(* Logix 5000 project; controller reports 1756-L63 rev 20.15; software revision 20.04; part 6 of 52 *)

        [520].time.Hour := 2, [520].time.Minute := 29, [520].time.Second := 59, [521].log_data[0].min := 1.0, [521].log_data[0].max := 1.0, [521].log_data[0].total := 900.0, [521].log_data[0].time := 900.0, [521].log_data[0].minminute := 30, [521].log_data[0].maxminute := 30, [521].log_data[0].valid := 1, [521].log_data[1].valid := 1, [521].log_data[2].valid := 1, [521].log_data[3].valid := 1, [521].log_data[4].valid := 1, [521].log_data[5].valid := 1, [521].log_data[6].valid := 1, [521].log_data[7].valid := 1, [521].log_data[8].valid := 1, [521].log_data[9].valid := 1, [521].log_data[10].valid := 1, [521].log_data[11].valid := 1, [521].log_data[12].valid := 1, [521].log_data[13].valid := 1, [521].log_data[14].valid := 1, [521].log_data[15].valid := 1, [521].log_data[16].valid := 1, [521].log_data[17].valid := 1, [521].log_data[18].valid := 1, [521].log_data[19].valid := 1, [521].time.Year := 2023, [521].time.Month := 1, [521].time.Day := 13, [521].time.Hour := 2, [521].time.Minute := 44, [521].time.Second := 59, [522].log_data[0].min := 1.0, [522].log_data[0].max := 1.0, [522].log_data[0].total := 900.0, [522].log_data[0].time := 900.0, [522].log_data[0].minminute := 45, [522].log_data[0].maxminute := 45, [522].log_data[0].valid := 1, [522].log_data[1].valid := 1, [522].log_data[2].valid := 1, [522].log_data[3].valid := 1, [522].log_data[4].valid := 1, [522].log_data[5].valid := 1, [522].log_data[6].valid := 1, [522].log_data[7].valid := 1, [522].log_data[8].valid := 1, [522].log_data[9].valid := 1, [522].log_data[10].valid := 1, [522].log_data[11].valid := 1, [522].log_data[12].valid := 1, [522].log_data[13].valid := 1, [522].log_data[14].valid := 1, [522].log_data[15].valid := 1, [522].log_data[16].valid := 1, [522].log_data[17].valid := 1, [522].log_data[18].valid := 1,
        [522].log_data[19].valid := 1, [522].time.Year := 2023, [522].time.Month := 1, [522].time.Day := 13, [522].time.Hour := 2, [522].time.Minute := 59, [522].time.Second := 59, [523].log_data[0].min := 1.0, [523].log_data[0].max := 1.0, [523].log_data[0].total := 900.0, [523].log_data[0].time := 900.0, [523].log_data[0].valid := 1, [523].log_data[1].valid := 1, [523].log_data[2].valid := 1, [523].log_data[3].valid := 1, [523].log_data[4].valid := 1, [523].log_data[5].valid := 1, [523].log_data[6].valid := 1, [523].log_data[7].valid := 1, [523].log_data[8].valid := 1, [523].log_data[9].valid := 1, [523].log_data[10].valid := 1, [523].log_data[11].valid := 1, [523].log_data[12].valid := 1, [523].log_data[13].valid := 1, [523].log_data[14].valid := 1, [523].log_data[15].valid := 1, [523].log_data[16].valid := 1, [523].log_data[17].valid := 1, [523].log_data[18].valid := 1, [523].log_data[19].valid := 1, [523].time.Year := 2023, [523].time.Month := 1, [523].time.Day := 13, [523].time.Hour := 3, [523].time.Minute := 14, [523].time.Second := 59, [524].log_data[0].min := 1.0, [524].log_data[0].max := 1.0, [524].log_data[0].total := 900.0, [524].log_data[0].time := 900.0, [524].log_data[0].minminute := 15, [524].log_data[0].maxminute := 15, [524].log_data[0].valid := 1, [524].log_data[1].valid := 1, [524].log_data[2].valid := 1, [524].log_data[3].valid := 1, [524].log_data[4].valid := 1, [524].log_data[5].valid := 1, [524].log_data[6].valid := 1, [524].log_data[7].valid := 1, [524].log_data[8].valid := 1, [524].log_data[9].valid := 1, [524].log_data[10].valid := 1, [524].log_data[11].valid := 1, [524].log_data[12].valid := 1, [524].log_data[13].valid := 1, [524].log_data[14].valid := 1, [524].log_data[15].valid := 1, [524].log_data[16].valid := 1,
        [524].log_data[17].valid := 1, [524].log_data[18].valid := 1, [524].log_data[19].valid := 1, [524].time.Year := 2023, [524].time.Month := 1, [524].time.Day := 13, [524].time.Hour := 3, [524].time.Minute := 29, [524].time.Second := 59, [525].log_data[0].min := 1.0, [525].log_data[0].max := 1.0, [525].log_data[0].total := 900.0, [525].log_data[0].time := 900.0, [525].log_data[0].minminute := 30, [525].log_data[0].maxminute := 30, [525].log_data[0].valid := 1, [525].log_data[1].valid := 1, [525].log_data[2].valid := 1, [525].log_data[3].valid := 1, [525].log_data[4].valid := 1, [525].log_data[5].valid := 1, [525].log_data[6].valid := 1, [525].log_data[7].valid := 1, [525].log_data[8].valid := 1, [525].log_data[9].valid := 1, [525].log_data[10].valid := 1, [525].log_data[11].valid := 1, [525].log_data[12].valid := 1, [525].log_data[13].valid := 1, [525].log_data[14].valid := 1, [525].log_data[15].valid := 1, [525].log_data[16].valid := 1, [525].log_data[17].valid := 1, [525].log_data[18].valid := 1, [525].log_data[19].valid := 1, [525].time.Year := 2023, [525].time.Month := 1, [525].time.Day := 13, [525].time.Hour := 3, [525].time.Minute := 44, [525].time.Second := 59, [526].log_data[0].min := 1.0, [526].log_data[0].max := 1.0, [526].log_data[0].total := 900.0, [526].log_data[0].time := 900.0, [526].log_data[0].minminute := 45, [526].log_data[0].maxminute := 45, [526].log_data[0].valid := 1, [526].log_data[1].valid := 1, [526].log_data[2].valid := 1, [526].log_data[3].valid := 1, [526].log_data[4].valid := 1, [526].log_data[5].valid := 1, [526].log_data[6].valid := 1, [526].log_data[7].valid := 1, [526].log_data[8].valid := 1, [526].log_data[9].valid := 1, [526].log_data[10].valid := 1, [526].log_data[11].valid := 1, [526].log_data[12].valid := 1,
        [526].log_data[13].valid := 1, [526].log_data[14].valid := 1, [526].log_data[15].valid := 1, [526].log_data[16].valid := 1, [526].log_data[17].valid := 1, [526].log_data[18].valid := 1, [526].log_data[19].valid := 1, [526].time.Year := 2023, [526].time.Month := 1, [526].time.Day := 13, [526].time.Hour := 3, [526].time.Minute := 59, [526].time.Second := 59, [527].log_data[0].min := 1.0, [527].log_data[0].max := 1.0, [527].log_data[0].total := 900.0, [527].log_data[0].time := 900.0, [527].log_data[0].valid := 1, [527].log_data[1].valid := 1, [527].log_data[2].valid := 1, [527].log_data[3].valid := 1, [527].log_data[4].valid := 1, [527].log_data[5].valid := 1, [527].log_data[6].valid := 1, [527].log_data[7].valid := 1, [527].log_data[8].valid := 1, [527].log_data[9].valid := 1, [527].log_data[10].valid := 1, [527].log_data[11].valid := 1, [527].log_data[12].valid := 1, [527].log_data[13].valid := 1, [527].log_data[14].valid := 1, [527].log_data[15].valid := 1, [527].log_data[16].valid := 1, [527].log_data[17].valid := 1, [527].log_data[18].valid := 1, [527].log_data[19].valid := 1, [527].time.Year := 2023, [527].time.Month := 1, [527].time.Day := 13, [527].time.Hour := 4, [527].time.Minute := 14, [527].time.Second := 59, [528].log_data[0].min := 1.0, [528].log_data[0].max := 1.0, [528].log_data[0].total := 900.0, [528].log_data[0].time := 900.0, [528].log_data[0].minminute := 15, [528].log_data[0].maxminute := 15, [528].log_data[0].valid := 1, [528].log_data[1].valid := 1, [528].log_data[2].valid := 1, [528].log_data[3].valid := 1, [528].log_data[4].valid := 1, [528].log_data[5].valid := 1, [528].log_data[6].valid := 1, [528].log_data[7].valid := 1, [528].log_data[8].valid := 1, [528].log_data[9].valid := 1, [528].log_data[10].valid := 1,
        [528].log_data[11].valid := 1, [528].log_data[12].valid := 1, [528].log_data[13].valid := 1, [528].log_data[14].valid := 1, [528].log_data[15].valid := 1, [528].log_data[16].valid := 1, [528].log_data[17].valid := 1, [528].log_data[18].valid := 1, [528].log_data[19].valid := 1, [528].time.Year := 2023, [528].time.Month := 1, [528].time.Day := 13, [528].time.Hour := 4, [528].time.Minute := 29, [528].time.Second := 59, [529].log_data[0].min := 1.0, [529].log_data[0].max := 1.0, [529].log_data[0].total := 900.0, [529].log_data[0].time := 900.0, [529].log_data[0].minminute := 30, [529].log_data[0].maxminute := 30, [529].log_data[0].valid := 1, [529].log_data[1].valid := 1, [529].log_data[2].valid := 1, [529].log_data[3].valid := 1, [529].log_data[4].valid := 1, [529].log_data[5].valid := 1, [529].log_data[6].valid := 1, [529].log_data[7].valid := 1, [529].log_data[8].valid := 1, [529].log_data[9].valid := 1, [529].log_data[10].valid := 1, [529].log_data[11].valid := 1, [529].log_data[12].valid := 1, [529].log_data[13].valid := 1, [529].log_data[14].valid := 1, [529].log_data[15].valid := 1, [529].log_data[16].valid := 1, [529].log_data[17].valid := 1, [529].log_data[18].valid := 1, [529].log_data[19].valid := 1, [529].time.Year := 2023, [529].time.Month := 1, [529].time.Day := 13, [529].time.Hour := 4, [529].time.Minute := 44, [529].time.Second := 59, [530].log_data[0].min := 1.0, [530].log_data[0].max := 1.0, [530].log_data[0].total := 900.0, [530].log_data[0].time := 900.0, [530].log_data[0].minminute := 45, [530].log_data[0].maxminute := 45, [530].log_data[0].valid := 1, [530].log_data[1].valid := 1, [530].log_data[2].valid := 1, [530].log_data[3].valid := 1, [530].log_data[4].valid := 1, [530].log_data[5].valid := 1, [530].log_data[6].valid := 1,
        [530].log_data[7].valid := 1, [530].log_data[8].valid := 1, [530].log_data[9].valid := 1, [530].log_data[10].valid := 1, [530].log_data[11].valid := 1, [530].log_data[12].valid := 1, [530].log_data[13].valid := 1, [530].log_data[14].valid := 1, [530].log_data[15].valid := 1, [530].log_data[16].valid := 1, [530].log_data[17].valid := 1, [530].log_data[18].valid := 1, [530].log_data[19].valid := 1, [530].time.Year := 2023, [530].time.Month := 1, [530].time.Day := 13, [530].time.Hour := 4, [530].time.Minute := 59, [530].time.Second := 59, [531].log_data[0].min := 1.0, [531].log_data[0].max := 1.0, [531].log_data[0].total := 900.0, [531].log_data[0].time := 900.0, [531].log_data[0].valid := 1, [531].log_data[1].valid := 1, [531].log_data[2].valid := 1, [531].log_data[3].valid := 1, [531].log_data[4].valid := 1, [531].log_data[5].valid := 1, [531].log_data[6].valid := 1, [531].log_data[7].valid := 1, [531].log_data[8].valid := 1, [531].log_data[9].valid := 1, [531].log_data[10].valid := 1, [531].log_data[11].valid := 1, [531].log_data[12].valid := 1, [531].log_data[13].valid := 1, [531].log_data[14].valid := 1, [531].log_data[15].valid := 1, [531].log_data[16].valid := 1, [531].log_data[17].valid := 1, [531].log_data[18].valid := 1, [531].log_data[19].valid := 1, [531].time.Year := 2023, [531].time.Month := 1, [531].time.Day := 13, [531].time.Hour := 5, [531].time.Minute := 14, [531].time.Second := 59, [532].log_data[0].min := 1.0, [532].log_data[0].max := 1.0, [532].log_data[0].total := 900.0, [532].log_data[0].time := 900.0, [532].log_data[0].minminute := 15, [532].log_data[0].maxminute := 15, [532].log_data[0].valid := 1, [532].log_data[1].valid := 1, [532].log_data[2].valid := 1, [532].log_data[3].valid := 1, [532].log_data[4].valid := 1,
        [532].log_data[5].valid := 1, [532].log_data[6].valid := 1, [532].log_data[7].valid := 1, [532].log_data[8].valid := 1, [532].log_data[9].valid := 1, [532].log_data[10].valid := 1, [532].log_data[11].valid := 1, [532].log_data[12].valid := 1, [532].log_data[13].valid := 1, [532].log_data[14].valid := 1, [532].log_data[15].valid := 1, [532].log_data[16].valid := 1, [532].log_data[17].valid := 1, [532].log_data[18].valid := 1, [532].log_data[19].valid := 1, [532].time.Year := 2023, [532].time.Month := 1, [532].time.Day := 13, [532].time.Hour := 5, [532].time.Minute := 29, [532].time.Second := 59, [533].log_data[0].min := 1.0, [533].log_data[0].max := 1.0, [533].log_data[0].total := 900.0, [533].log_data[0].time := 900.0, [533].log_data[0].minminute := 30, [533].log_data[0].maxminute := 30, [533].log_data[0].valid := 1, [533].log_data[1].valid := 1, [533].log_data[2].valid := 1, [533].log_data[3].valid := 1, [533].log_data[4].valid := 1, [533].log_data[5].valid := 1, [533].log_data[6].valid := 1, [533].log_data[7].valid := 1, [533].log_data[8].valid := 1, [533].log_data[9].valid := 1, [533].log_data[10].valid := 1, [533].log_data[11].valid := 1, [533].log_data[12].valid := 1, [533].log_data[13].valid := 1, [533].log_data[14].valid := 1, [533].log_data[15].valid := 1, [533].log_data[16].valid := 1, [533].log_data[17].valid := 1, [533].log_data[18].valid := 1, [533].log_data[19].valid := 1, [533].time.Year := 2023, [533].time.Month := 1, [533].time.Day := 13, [533].time.Hour := 5, [533].time.Minute := 44, [533].time.Second := 59, [534].log_data[0].min := 1.0, [534].log_data[0].max := 1.0, [534].log_data[0].total := 900.0, [534].log_data[0].time := 900.0, [534].log_data[0].minminute := 45, [534].log_data[0].maxminute := 45, [534].log_data[0].valid := 1,
        [534].log_data[1].valid := 1, [534].log_data[2].valid := 1, [534].log_data[3].valid := 1, [534].log_data[4].valid := 1, [534].log_data[5].valid := 1, [534].log_data[6].valid := 1, [534].log_data[7].valid := 1, [534].log_data[8].valid := 1, [534].log_data[9].valid := 1, [534].log_data[10].valid := 1, [534].log_data[11].valid := 1, [534].log_data[12].valid := 1, [534].log_data[13].valid := 1, [534].log_data[14].valid := 1, [534].log_data[15].valid := 1, [534].log_data[16].valid := 1, [534].log_data[17].valid := 1, [534].log_data[18].valid := 1, [534].log_data[19].valid := 1, [534].time.Year := 2023, [534].time.Month := 1, [534].time.Day := 13, [534].time.Hour := 5, [534].time.Minute := 59, [534].time.Second := 59, [535].log_data[0].min := 1.0, [535].log_data[0].max := 1.0, [535].log_data[0].total := 900.0, [535].log_data[0].time := 900.0, [535].log_data[0].valid := 1, [535].log_data[1].valid := 1, [535].log_data[2].valid := 1, [535].log_data[3].valid := 1, [535].log_data[4].valid := 1, [535].log_data[5].valid := 1, [535].log_data[6].valid := 1, [535].log_data[7].valid := 1, [535].log_data[8].valid := 1, [535].log_data[9].valid := 1, [535].log_data[10].valid := 1, [535].log_data[11].valid := 1, [535].log_data[12].valid := 1, [535].log_data[13].valid := 1, [535].log_data[14].valid := 1, [535].log_data[15].valid := 1, [535].log_data[16].valid := 1, [535].log_data[17].valid := 1, [535].log_data[18].valid := 1, [535].log_data[19].valid := 1, [535].time.Year := 2023, [535].time.Month := 1, [535].time.Day := 13, [535].time.Hour := 6, [535].time.Minute := 14, [535].time.Second := 59, [536].log_data[0].min := 1.0, [536].log_data[0].max := 1.0, [536].log_data[0].total := 900.0, [536].log_data[0].time := 900.0, [536].log_data[0].minminute := 15,
        [536].log_data[0].maxminute := 15, [536].log_data[0].valid := 1, [536].log_data[1].valid := 1, [536].log_data[2].valid := 1, [536].log_data[3].valid := 1, [536].log_data[4].valid := 1, [536].log_data[5].valid := 1, [536].log_data[6].valid := 1, [536].log_data[7].valid := 1, [536].log_data[8].valid := 1, [536].log_data[9].valid := 1, [536].log_data[10].valid := 1, [536].log_data[11].valid := 1, [536].log_data[12].valid := 1, [536].log_data[13].valid := 1, [536].log_data[14].valid := 1, [536].log_data[15].valid := 1, [536].log_data[16].valid := 1, [536].log_data[17].valid := 1, [536].log_data[18].valid := 1, [536].log_data[19].valid := 1, [536].time.Year := 2023, [536].time.Month := 1, [536].time.Day := 13, [536].time.Hour := 6, [536].time.Minute := 29, [536].time.Second := 59, [537].log_data[0].min := 1.0, [537].log_data[0].max := 1.0, [537].log_data[0].total := 900.0, [537].log_data[0].time := 900.0, [537].log_data[0].minminute := 30, [537].log_data[0].maxminute := 30, [537].log_data[0].valid := 1, [537].log_data[1].valid := 1, [537].log_data[2].valid := 1, [537].log_data[3].valid := 1, [537].log_data[4].valid := 1, [537].log_data[5].valid := 1, [537].log_data[6].valid := 1, [537].log_data[7].valid := 1, [537].log_data[8].valid := 1, [537].log_data[9].valid := 1, [537].log_data[10].valid := 1, [537].log_data[11].valid := 1, [537].log_data[12].valid := 1, [537].log_data[13].valid := 1, [537].log_data[14].valid := 1, [537].log_data[15].valid := 1, [537].log_data[16].valid := 1, [537].log_data[17].valid := 1, [537].log_data[18].valid := 1, [537].log_data[19].valid := 1, [537].time.Year := 2023, [537].time.Month := 1, [537].time.Day := 13, [537].time.Hour := 6, [537].time.Minute := 44, [537].time.Second := 59, [538].log_data[0].min := 1.0,
        [538].log_data[0].max := 1.0, [538].log_data[0].total := 900.0, [538].log_data[0].time := 900.0, [538].log_data[0].minminute := 45, [538].log_data[0].maxminute := 45, [538].log_data[0].valid := 1, [538].log_data[1].valid := 1, [538].log_data[2].valid := 1, [538].log_data[3].valid := 1, [538].log_data[4].valid := 1, [538].log_data[5].valid := 1, [538].log_data[6].valid := 1, [538].log_data[7].valid := 1, [538].log_data[8].valid := 1, [538].log_data[9].valid := 1, [538].log_data[10].valid := 1, [538].log_data[11].valid := 1, [538].log_data[12].valid := 1, [538].log_data[13].valid := 1, [538].log_data[14].valid := 1, [538].log_data[15].valid := 1, [538].log_data[16].valid := 1, [538].log_data[17].valid := 1, [538].log_data[18].valid := 1, [538].log_data[19].valid := 1, [538].time.Year := 2023, [538].time.Month := 1, [538].time.Day := 13, [538].time.Hour := 6, [538].time.Minute := 59, [538].time.Second := 59, [539].log_data[0].min := 1.0, [539].log_data[0].max := 1.0, [539].log_data[0].total := 900.0, [539].log_data[0].time := 900.0, [539].log_data[0].valid := 1, [539].log_data[1].valid := 1, [539].log_data[2].valid := 1, [539].log_data[3].valid := 1, [539].log_data[4].valid := 1, [539].log_data[5].valid := 1, [539].log_data[6].valid := 1, [539].log_data[7].valid := 1, [539].log_data[8].valid := 1, [539].log_data[9].valid := 1, [539].log_data[10].valid := 1, [539].log_data[11].valid := 1, [539].log_data[12].valid := 1, [539].log_data[13].valid := 1, [539].log_data[14].valid := 1, [539].log_data[15].valid := 1, [539].log_data[16].valid := 1, [539].log_data[17].valid := 1, [539].log_data[18].valid := 1, [539].log_data[19].valid := 1, [539].time.Year := 2023, [539].time.Month := 1, [539].time.Day := 13, [539].time.Hour := 7, [539].time.Minute := 14,
        [539].time.Second := 59, [540].log_data[0].min := 1.0, [540].log_data[0].max := 1.0, [540].log_data[0].total := 900.0, [540].log_data[0].time := 900.0, [540].log_data[0].minminute := 15, [540].log_data[0].maxminute := 15, [540].log_data[0].valid := 1, [540].log_data[1].valid := 1, [540].log_data[2].valid := 1, [540].log_data[3].valid := 1, [540].log_data[4].valid := 1, [540].log_data[5].valid := 1, [540].log_data[6].valid := 1, [540].log_data[7].valid := 1, [540].log_data[8].valid := 1, [540].log_data[9].valid := 1, [540].log_data[10].valid := 1, [540].log_data[11].valid := 1, [540].log_data[12].valid := 1, [540].log_data[13].valid := 1, [540].log_data[14].valid := 1, [540].log_data[15].valid := 1, [540].log_data[16].valid := 1, [540].log_data[17].valid := 1, [540].log_data[18].valid := 1, [540].log_data[19].valid := 1, [540].time.Year := 2023, [540].time.Month := 1, [540].time.Day := 13, [540].time.Hour := 7, [540].time.Minute := 29, [540].time.Second := 59, [541].log_data[0].min := 1.0, [541].log_data[0].max := 1.0, [541].log_data[0].total := 900.0, [541].log_data[0].time := 900.0, [541].log_data[0].minminute := 30, [541].log_data[0].maxminute := 30, [541].log_data[0].valid := 1, [541].log_data[1].valid := 1, [541].log_data[2].valid := 1, [541].log_data[3].valid := 1, [541].log_data[4].valid := 1, [541].log_data[5].valid := 1, [541].log_data[6].valid := 1, [541].log_data[7].valid := 1, [541].log_data[8].valid := 1, [541].log_data[9].valid := 1, [541].log_data[10].valid := 1, [541].log_data[11].valid := 1, [541].log_data[12].valid := 1, [541].log_data[13].valid := 1, [541].log_data[14].valid := 1, [541].log_data[15].valid := 1, [541].log_data[16].valid := 1, [541].log_data[17].valid := 1, [541].log_data[18].valid := 1, [541].log_data[19].valid := 1, [541].time.Year := 2023,
        [541].time.Month := 1, [541].time.Day := 13, [541].time.Hour := 7, [541].time.Minute := 44, [541].time.Second := 59, [542].log_data[0].min := 1.0, [542].log_data[0].max := 1.0, [542].log_data[0].total := 900.0, [542].log_data[0].time := 900.0, [542].log_data[0].minminute := 45, [542].log_data[0].maxminute := 45, [542].log_data[0].valid := 1, [542].log_data[1].valid := 1, [542].log_data[2].valid := 1, [542].log_data[3].valid := 1, [542].log_data[4].valid := 1, [542].log_data[5].valid := 1, [542].log_data[6].valid := 1, [542].log_data[7].valid := 1, [542].log_data[8].valid := 1, [542].log_data[9].valid := 1, [542].log_data[10].valid := 1, [542].log_data[11].valid := 1, [542].log_data[12].valid := 1, [542].log_data[13].valid := 1, [542].log_data[14].valid := 1, [542].log_data[15].valid := 1, [542].log_data[16].valid := 1, [542].log_data[17].valid := 1, [542].log_data[18].valid := 1, [542].log_data[19].valid := 1, [542].time.Year := 2023, [542].time.Month := 1, [542].time.Day := 13, [542].time.Hour := 7, [542].time.Minute := 59, [542].time.Second := 59, [543].log_data[0].min := 1.0, [543].log_data[0].max := 1.0, [543].log_data[0].total := 900.0, [543].log_data[0].time := 900.0, [543].log_data[0].valid := 1, [543].log_data[1].valid := 1, [543].log_data[2].valid := 1, [543].log_data[3].valid := 1, [543].log_data[4].valid := 1, [543].log_data[5].valid := 1, [543].log_data[6].valid := 1, [543].log_data[7].valid := 1, [543].log_data[8].valid := 1, [543].log_data[9].valid := 1, [543].log_data[10].valid := 1, [543].log_data[11].valid := 1, [543].log_data[12].valid := 1, [543].log_data[13].valid := 1, [543].log_data[14].valid := 1, [543].log_data[15].valid := 1, [543].log_data[16].valid := 1, [543].log_data[17].valid := 1, [543].log_data[18].valid := 1,
        [543].log_data[19].valid := 1, [543].time.Year := 2023, [543].time.Month := 1, [543].time.Day := 13, [543].time.Hour := 8, [543].time.Minute := 14, [543].time.Second := 59, [544].log_data[0].min := 1.0, [544].log_data[0].max := 1.0, [544].log_data[0].total := 900.0, [544].log_data[0].time := 900.0, [544].log_data[0].minminute := 15, [544].log_data[0].maxminute := 15, [544].log_data[0].valid := 1, [544].log_data[1].valid := 1, [544].log_data[2].valid := 1, [544].log_data[3].valid := 1, [544].log_data[4].valid := 1, [544].log_data[5].valid := 1, [544].log_data[6].valid := 1, [544].log_data[7].valid := 1, [544].log_data[8].valid := 1, [544].log_data[9].valid := 1, [544].log_data[10].valid := 1, [544].log_data[11].valid := 1, [544].log_data[12].valid := 1, [544].log_data[13].valid := 1, [544].log_data[14].valid := 1, [544].log_data[15].valid := 1, [544].log_data[16].valid := 1, [544].log_data[17].valid := 1, [544].log_data[18].valid := 1, [544].log_data[19].valid := 1, [544].time.Year := 2023, [544].time.Month := 1, [544].time.Day := 13, [544].time.Hour := 8, [544].time.Minute := 29, [544].time.Second := 59, [545].log_data[0].min := 1.0, [545].log_data[0].max := 1.0, [545].log_data[0].total := 900.0, [545].log_data[0].time := 900.0, [545].log_data[0].minminute := 30, [545].log_data[0].maxminute := 30, [545].log_data[0].valid := 1, [545].log_data[1].valid := 1, [545].log_data[2].valid := 1, [545].log_data[3].valid := 1, [545].log_data[4].valid := 1, [545].log_data[5].valid := 1, [545].log_data[6].valid := 1, [545].log_data[7].valid := 1, [545].log_data[8].valid := 1, [545].log_data[9].valid := 1, [545].log_data[10].valid := 1, [545].log_data[11].valid := 1, [545].log_data[12].valid := 1, [545].log_data[13].valid := 1, [545].log_data[14].valid := 1,
        [545].log_data[15].valid := 1, [545].log_data[16].valid := 1, [545].log_data[17].valid := 1, [545].log_data[18].valid := 1, [545].log_data[19].valid := 1, [545].time.Year := 2023, [545].time.Month := 1, [545].time.Day := 13, [545].time.Hour := 8, [545].time.Minute := 44, [545].time.Second := 59, [546].log_data[0].min := 1.0, [546].log_data[0].max := 1.0, [546].log_data[0].total := 900.0, [546].log_data[0].time := 900.0, [546].log_data[0].minminute := 45, [546].log_data[0].maxminute := 45, [546].log_data[0].valid := 1, [546].log_data[1].valid := 1, [546].log_data[2].valid := 1, [546].log_data[3].valid := 1, [546].log_data[4].valid := 1, [546].log_data[5].valid := 1, [546].log_data[6].valid := 1, [546].log_data[7].valid := 1, [546].log_data[8].valid := 1, [546].log_data[9].valid := 1, [546].log_data[10].valid := 1, [546].log_data[11].valid := 1, [546].log_data[12].valid := 1, [546].log_data[13].valid := 1, [546].log_data[14].valid := 1, [546].log_data[15].valid := 1, [546].log_data[16].valid := 1, [546].log_data[17].valid := 1, [546].log_data[18].valid := 1, [546].log_data[19].valid := 1, [546].time.Year := 2023, [546].time.Month := 1, [546].time.Day := 13, [546].time.Hour := 8, [546].time.Minute := 59, [546].time.Second := 59, [547].log_data[0].min := 1.0, [547].log_data[0].max := 1.0, [547].log_data[0].total := 900.0, [547].log_data[0].time := 900.0, [547].log_data[0].valid := 1, [547].log_data[1].valid := 1, [547].log_data[2].valid := 1, [547].log_data[3].valid := 1, [547].log_data[4].valid := 1, [547].log_data[5].valid := 1, [547].log_data[6].valid := 1, [547].log_data[7].valid := 1, [547].log_data[8].valid := 1, [547].log_data[9].valid := 1, [547].log_data[10].valid := 1, [547].log_data[11].valid := 1, [547].log_data[12].valid := 1,
        [547].log_data[13].valid := 1, [547].log_data[14].valid := 1, [547].log_data[15].valid := 1, [547].log_data[16].valid := 1, [547].log_data[17].valid := 1, [547].log_data[18].valid := 1, [547].log_data[19].valid := 1, [547].time.Year := 2023, [547].time.Month := 1, [547].time.Day := 13, [547].time.Hour := 9, [547].time.Minute := 14, [547].time.Second := 59, [548].log_data[0].min := 1.0, [548].log_data[0].max := 1.0, [548].log_data[0].total := 900.0, [548].log_data[0].time := 900.0, [548].log_data[0].minminute := 15, [548].log_data[0].maxminute := 15, [548].log_data[0].valid := 1, [548].log_data[1].valid := 1, [548].log_data[2].valid := 1, [548].log_data[3].valid := 1, [548].log_data[4].valid := 1, [548].log_data[5].valid := 1, [548].log_data[6].valid := 1, [548].log_data[7].valid := 1, [548].log_data[8].valid := 1, [548].log_data[9].valid := 1, [548].log_data[10].valid := 1, [548].log_data[11].valid := 1, [548].log_data[12].valid := 1, [548].log_data[13].valid := 1, [548].log_data[14].valid := 1, [548].log_data[15].valid := 1, [548].log_data[16].valid := 1, [548].log_data[17].valid := 1, [548].log_data[18].valid := 1, [548].log_data[19].valid := 1, [548].time.Year := 2023, [548].time.Month := 1, [548].time.Day := 13, [548].time.Hour := 9, [548].time.Minute := 29, [548].time.Second := 59, [549].log_data[0].min := 1.0, [549].log_data[0].max := 1.0, [549].log_data[0].total := 900.0, [549].log_data[0].time := 900.0, [549].log_data[0].minminute := 30, [549].log_data[0].maxminute := 30, [549].log_data[0].valid := 1, [549].log_data[1].valid := 1, [549].log_data[2].valid := 1, [549].log_data[3].valid := 1, [549].log_data[4].valid := 1, [549].log_data[5].valid := 1, [549].log_data[6].valid := 1, [549].log_data[7].valid := 1, [549].log_data[8].valid := 1,
        [549].log_data[9].valid := 1, [549].log_data[10].valid := 1, [549].log_data[11].valid := 1, [549].log_data[12].valid := 1, [549].log_data[13].valid := 1, [549].log_data[14].valid := 1, [549].log_data[15].valid := 1, [549].log_data[16].valid := 1, [549].log_data[17].valid := 1, [549].log_data[18].valid := 1, [549].log_data[19].valid := 1, [549].time.Year := 2023, [549].time.Month := 1, [549].time.Day := 13, [549].time.Hour := 9, [549].time.Minute := 44, [549].time.Second := 59, [550].log_data[0].min := 1.0, [550].log_data[0].max := 1.0, [550].log_data[0].total := 900.0, [550].log_data[0].time := 900.0, [550].log_data[0].minminute := 45, [550].log_data[0].maxminute := 45, [550].log_data[0].valid := 1, [550].log_data[1].valid := 1, [550].log_data[2].valid := 1, [550].log_data[3].valid := 1, [550].log_data[4].valid := 1, [550].log_data[5].valid := 1, [550].log_data[6].valid := 1, [550].log_data[7].valid := 1, [550].log_data[8].valid := 1, [550].log_data[9].valid := 1, [550].log_data[10].valid := 1, [550].log_data[11].valid := 1, [550].log_data[12].valid := 1, [550].log_data[13].valid := 1, [550].log_data[14].valid := 1, [550].log_data[15].valid := 1, [550].log_data[16].valid := 1, [550].log_data[17].valid := 1, [550].log_data[18].valid := 1, [550].log_data[19].valid := 1, [550].time.Year := 2023, [550].time.Month := 1, [550].time.Day := 13, [550].time.Hour := 9, [550].time.Minute := 59, [550].time.Second := 59, [551].log_data[0].min := 1.0, [551].log_data[0].max := 1.0, [551].log_data[0].total := 900.0, [551].log_data[0].time := 900.0, [551].log_data[0].valid := 1, [551].log_data[1].valid := 1, [551].log_data[2].valid := 1, [551].log_data[3].valid := 1, [551].log_data[4].valid := 1, [551].log_data[5].valid := 1, [551].log_data[6].valid := 1,
        [551].log_data[7].valid := 1, [551].log_data[8].valid := 1, [551].log_data[9].valid := 1, [551].log_data[10].valid := 1, [551].log_data[11].valid := 1, [551].log_data[12].valid := 1, [551].log_data[13].valid := 1, [551].log_data[14].valid := 1, [551].log_data[15].valid := 1, [551].log_data[16].valid := 1, [551].log_data[17].valid := 1, [551].log_data[18].valid := 1, [551].log_data[19].valid := 1, [551].time.Year := 2023, [551].time.Month := 1, [551].time.Day := 13, [551].time.Hour := 10, [551].time.Minute := 14, [551].time.Second := 59, [552].log_data[0].min := 1.0, [552].log_data[0].max := 1.0, [552].log_data[0].total := 900.0, [552].log_data[0].time := 900.0, [552].log_data[0].minminute := 15, [552].log_data[0].maxminute := 15, [552].log_data[0].valid := 1, [552].log_data[1].valid := 1, [552].log_data[2].valid := 1, [552].log_data[3].valid := 1, [552].log_data[4].valid := 1, [552].log_data[5].valid := 1, [552].log_data[6].valid := 1, [552].log_data[7].valid := 1, [552].log_data[8].valid := 1, [552].log_data[9].valid := 1, [552].log_data[10].valid := 1, [552].log_data[11].valid := 1, [552].log_data[12].valid := 1, [552].log_data[13].valid := 1, [552].log_data[14].valid := 1, [552].log_data[15].valid := 1, [552].log_data[16].valid := 1, [552].log_data[17].valid := 1, [552].log_data[18].valid := 1, [552].log_data[19].valid := 1, [552].time.Year := 2023, [552].time.Month := 1, [552].time.Day := 13, [552].time.Hour := 10, [552].time.Minute := 29, [552].time.Second := 59, [553].log_data[0].min := 1.0, [553].log_data[0].max := 1.0, [553].log_data[0].total := 900.0, [553].log_data[0].time := 900.0, [553].log_data[0].minminute := 30, [553].log_data[0].maxminute := 30, [553].log_data[0].valid := 1, [553].log_data[1].valid := 1, [553].log_data[2].valid := 1,
        [553].log_data[3].valid := 1, [553].log_data[4].valid := 1, [553].log_data[5].valid := 1, [553].log_data[6].valid := 1, [553].log_data[7].valid := 1, [553].log_data[8].valid := 1, [553].log_data[9].valid := 1, [553].log_data[10].valid := 1, [553].log_data[11].valid := 1, [553].log_data[12].valid := 1, [553].log_data[13].valid := 1, [553].log_data[14].valid := 1, [553].log_data[15].valid := 1, [553].log_data[16].valid := 1, [553].log_data[17].valid := 1, [553].log_data[18].valid := 1, [553].log_data[19].valid := 1, [553].time.Year := 2023, [553].time.Month := 1, [553].time.Day := 13, [553].time.Hour := 10, [553].time.Minute := 44, [553].time.Second := 59, [554].log_data[0].min := 1.0, [554].log_data[0].max := 1.0, [554].log_data[0].total := 900.0, [554].log_data[0].time := 900.0, [554].log_data[0].minminute := 45, [554].log_data[0].maxminute := 45, [554].log_data[0].valid := 1, [554].log_data[1].valid := 1, [554].log_data[2].valid := 1, [554].log_data[3].valid := 1, [554].log_data[4].valid := 1, [554].log_data[5].valid := 1, [554].log_data[6].valid := 1, [554].log_data[7].valid := 1, [554].log_data[8].valid := 1, [554].log_data[9].valid := 1, [554].log_data[10].valid := 1, [554].log_data[11].valid := 1, [554].log_data[12].valid := 1, [554].log_data[13].valid := 1, [554].log_data[14].valid := 1, [554].log_data[15].valid := 1, [554].log_data[16].valid := 1, [554].log_data[17].valid := 1, [554].log_data[18].valid := 1, [554].log_data[19].valid := 1, [554].time.Year := 2023, [554].time.Month := 1, [554].time.Day := 13, [554].time.Hour := 10, [554].time.Minute := 59, [554].time.Second := 59, [555].log_data[0].min := 1.0, [555].log_data[0].max := 1.0, [555].log_data[0].total := 900.0, [555].log_data[0].time := 900.0, [555].log_data[0].valid := 1,
        [555].log_data[1].valid := 1, [555].log_data[2].valid := 1, [555].log_data[3].valid := 1, [555].log_data[4].valid := 1, [555].log_data[5].valid := 1, [555].log_data[6].valid := 1, [555].log_data[7].valid := 1, [555].log_data[8].valid := 1, [555].log_data[9].valid := 1, [555].log_data[10].valid := 1, [555].log_data[11].valid := 1, [555].log_data[12].valid := 1, [555].log_data[13].valid := 1, [555].log_data[14].valid := 1, [555].log_data[15].valid := 1, [555].log_data[16].valid := 1, [555].log_data[17].valid := 1, [555].log_data[18].valid := 1, [555].log_data[19].valid := 1, [555].time.Year := 2023, [555].time.Month := 1, [555].time.Day := 13, [555].time.Hour := 11, [555].time.Minute := 14, [555].time.Second := 59, [556].log_data[0].min := 1.0, [556].log_data[0].max := 1.0, [556].log_data[0].total := 900.0, [556].log_data[0].time := 900.0, [556].log_data[0].minminute := 15, [556].log_data[0].maxminute := 15, [556].log_data[0].valid := 1, [556].log_data[1].valid := 1, [556].log_data[2].valid := 1, [556].log_data[3].valid := 1, [556].log_data[4].valid := 1, [556].log_data[5].valid := 1, [556].log_data[6].valid := 1, [556].log_data[7].valid := 1, [556].log_data[8].valid := 1, [556].log_data[9].valid := 1, [556].log_data[10].valid := 1, [556].log_data[11].valid := 1, [556].log_data[12].valid := 1, [556].log_data[13].valid := 1, [556].log_data[14].valid := 1, [556].log_data[15].valid := 1, [556].log_data[16].valid := 1, [556].log_data[17].valid := 1, [556].log_data[18].valid := 1, [556].log_data[19].valid := 1, [556].time.Year := 2023, [556].time.Month := 1, [556].time.Day := 13, [556].time.Hour := 11, [556].time.Minute := 29, [556].time.Second := 59, [557].log_data[0].min := 1.0, [557].log_data[0].max := 1.0, [557].log_data[0].total := 900.0,
        [557].log_data[0].time := 900.0, [557].log_data[0].minminute := 30, [557].log_data[0].maxminute := 30, [557].log_data[0].valid := 1, [557].log_data[1].valid := 1, [557].log_data[2].valid := 1, [557].log_data[3].valid := 1, [557].log_data[4].valid := 1, [557].log_data[5].valid := 1, [557].log_data[6].valid := 1, [557].log_data[7].valid := 1, [557].log_data[8].valid := 1, [557].log_data[9].valid := 1, [557].log_data[10].valid := 1, [557].log_data[11].valid := 1, [557].log_data[12].valid := 1, [557].log_data[13].valid := 1, [557].log_data[14].valid := 1, [557].log_data[15].valid := 1, [557].log_data[16].valid := 1, [557].log_data[17].valid := 1, [557].log_data[18].valid := 1, [557].log_data[19].valid := 1, [557].time.Year := 2023, [557].time.Month := 1, [557].time.Day := 13, [557].time.Hour := 11, [557].time.Minute := 44, [557].time.Second := 59, [558].log_data[0].min := 1.0, [558].log_data[0].max := 1.0, [558].log_data[0].total := 900.0, [558].log_data[0].time := 900.0, [558].log_data[0].minminute := 45, [558].log_data[0].maxminute := 45, [558].log_data[0].valid := 1, [558].log_data[1].valid := 1, [558].log_data[2].valid := 1, [558].log_data[3].valid := 1, [558].log_data[4].valid := 1, [558].log_data[5].valid := 1, [558].log_data[6].valid := 1, [558].log_data[7].valid := 1, [558].log_data[8].valid := 1, [558].log_data[9].valid := 1, [558].log_data[10].valid := 1, [558].log_data[11].valid := 1, [558].log_data[12].valid := 1, [558].log_data[13].valid := 1, [558].log_data[14].valid := 1, [558].log_data[15].valid := 1, [558].log_data[16].valid := 1, [558].log_data[17].valid := 1, [558].log_data[18].valid := 1, [558].log_data[19].valid := 1, [558].time.Year := 2023, [558].time.Month := 1, [558].time.Day := 13, [558].time.Hour := 11, [558].time.Minute := 59,
        [558].time.Second := 59, [559].log_data[0].min := 1.0, [559].log_data[0].max := 1.0, [559].log_data[0].total := 900.0, [559].log_data[0].time := 900.0, [559].log_data[0].valid := 1, [559].log_data[1].valid := 1, [559].log_data[2].valid := 1, [559].log_data[3].valid := 1, [559].log_data[4].valid := 1, [559].log_data[5].valid := 1, [559].log_data[6].valid := 1, [559].log_data[7].valid := 1, [559].log_data[8].valid := 1, [559].log_data[9].valid := 1, [559].log_data[10].valid := 1, [559].log_data[11].valid := 1, [559].log_data[12].valid := 1, [559].log_data[13].valid := 1, [559].log_data[14].valid := 1, [559].log_data[15].valid := 1, [559].log_data[16].valid := 1, [559].log_data[17].valid := 1, [559].log_data[18].valid := 1, [559].log_data[19].valid := 1, [559].time.Year := 2023, [559].time.Month := 1, [559].time.Day := 13, [559].time.Hour := 12, [559].time.Minute := 14, [559].time.Second := 59, [560].log_data[0].min := 1.0, [560].log_data[0].max := 1.0, [560].log_data[0].total := 900.0, [560].log_data[0].time := 900.0, [560].log_data[0].minminute := 15, [560].log_data[0].maxminute := 15, [560].log_data[0].valid := 1, [560].log_data[1].valid := 1, [560].log_data[2].valid := 1, [560].log_data[3].valid := 1, [560].log_data[4].valid := 1, [560].log_data[5].valid := 1, [560].log_data[6].valid := 1, [560].log_data[7].valid := 1, [560].log_data[8].valid := 1, [560].log_data[9].valid := 1, [560].log_data[10].valid := 1, [560].log_data[11].valid := 1, [560].log_data[12].valid := 1, [560].log_data[13].valid := 1, [560].log_data[14].valid := 1, [560].log_data[15].valid := 1, [560].log_data[16].valid := 1, [560].log_data[17].valid := 1, [560].log_data[18].valid := 1, [560].log_data[19].valid := 1, [560].time.Year := 2023, [560].time.Month := 1, [560].time.Day := 13,
        [560].time.Hour := 12, [560].time.Minute := 29, [560].time.Second := 59, [561].log_data[0].min := 1.0, [561].log_data[0].max := 1.0, [561].log_data[0].total := 900.0, [561].log_data[0].time := 900.0, [561].log_data[0].minminute := 30, [561].log_data[0].maxminute := 30, [561].log_data[0].valid := 1, [561].log_data[1].valid := 1, [561].log_data[2].valid := 1, [561].log_data[3].valid := 1, [561].log_data[4].valid := 1, [561].log_data[5].valid := 1, [561].log_data[6].valid := 1, [561].log_data[7].valid := 1, [561].log_data[8].valid := 1, [561].log_data[9].valid := 1, [561].log_data[10].valid := 1, [561].log_data[11].valid := 1, [561].log_data[12].valid := 1, [561].log_data[13].valid := 1, [561].log_data[14].valid := 1, [561].log_data[15].valid := 1, [561].log_data[16].valid := 1, [561].log_data[17].valid := 1, [561].log_data[18].valid := 1, [561].log_data[19].valid := 1, [561].time.Year := 2023, [561].time.Month := 1, [561].time.Day := 13, [561].time.Hour := 12, [561].time.Minute := 44, [561].time.Second := 59, [562].log_data[0].min := 1.0, [562].log_data[0].max := 1.0, [562].log_data[0].total := 900.0, [562].log_data[0].time := 900.0, [562].log_data[0].minminute := 45, [562].log_data[0].maxminute := 45, [562].log_data[0].valid := 1, [562].log_data[1].valid := 1, [562].log_data[2].valid := 1, [562].log_data[3].valid := 1, [562].log_data[4].valid := 1, [562].log_data[5].valid := 1, [562].log_data[6].valid := 1, [562].log_data[7].valid := 1, [562].log_data[8].valid := 1, [562].log_data[9].valid := 1, [562].log_data[10].valid := 1, [562].log_data[11].valid := 1, [562].log_data[12].valid := 1, [562].log_data[13].valid := 1, [562].log_data[14].valid := 1, [562].log_data[15].valid := 1, [562].log_data[16].valid := 1, [562].log_data[17].valid := 1, [562].log_data[18].valid := 1,
        [562].log_data[19].valid := 1, [562].time.Year := 2023, [562].time.Month := 1, [562].time.Day := 13, [562].time.Hour := 12, [562].time.Minute := 59, [562].time.Second := 59, [563].log_data[0].min := 1.0, [563].log_data[0].max := 1.0, [563].log_data[0].total := 899.5, [563].log_data[0].time := 899.5, [563].log_data[0].valid := 1, [563].log_data[1].valid := 1, [563].log_data[2].valid := 1, [563].log_data[3].valid := 1, [563].log_data[4].valid := 1, [563].log_data[5].valid := 1, [563].log_data[6].valid := 1, [563].log_data[7].valid := 1, [563].log_data[8].valid := 1, [563].log_data[9].valid := 1, [563].log_data[10].valid := 1, [563].log_data[11].valid := 1, [563].log_data[12].valid := 1, [563].log_data[13].valid := 1, [563].log_data[14].valid := 1, [563].log_data[15].valid := 1, [563].log_data[16].valid := 1, [563].log_data[17].valid := 1, [563].log_data[18].valid := 1, [563].log_data[19].valid := 1, [563].time.Year := 2023, [563].time.Month := 1, [563].time.Day := 13, [563].time.Hour := 13, [563].time.Minute := 14, [563].time.Second := 59, [564].log_data[0].min := 1.0, [564].log_data[0].max := 1.0, [564].log_data[0].total := 900.0, [564].log_data[0].time := 900.0, [564].log_data[0].minminute := 15, [564].log_data[0].maxminute := 15, [564].log_data[0].valid := 1, [564].log_data[1].valid := 1, [564].log_data[2].valid := 1, [564].log_data[3].valid := 1, [564].log_data[4].valid := 1, [564].log_data[5].valid := 1, [564].log_data[6].valid := 1, [564].log_data[7].valid := 1, [564].log_data[8].valid := 1, [564].log_data[9].valid := 1, [564].log_data[10].valid := 1, [564].log_data[11].valid := 1, [564].log_data[12].valid := 1, [564].log_data[13].valid := 1, [564].log_data[14].valid := 1, [564].log_data[15].valid := 1, [564].log_data[16].valid := 1,
        [564].log_data[17].valid := 1, [564].log_data[18].valid := 1, [564].log_data[19].valid := 1, [564].time.Year := 2023, [564].time.Month := 1, [564].time.Day := 13, [564].time.Hour := 13, [564].time.Minute := 29, [564].time.Second := 59, [565].log_data[0].min := 1.0, [565].log_data[0].max := 1.0, [565].log_data[0].total := 900.0, [565].log_data[0].time := 900.0, [565].log_data[0].minminute := 30, [565].log_data[0].maxminute := 30, [565].log_data[0].valid := 1, [565].log_data[1].valid := 1, [565].log_data[2].valid := 1, [565].log_data[3].valid := 1, [565].log_data[4].valid := 1, [565].log_data[5].valid := 1, [565].log_data[6].valid := 1, [565].log_data[7].valid := 1, [565].log_data[8].valid := 1, [565].log_data[9].valid := 1, [565].log_data[10].valid := 1, [565].log_data[11].valid := 1, [565].log_data[12].valid := 1, [565].log_data[13].valid := 1, [565].log_data[14].valid := 1, [565].log_data[15].valid := 1, [565].log_data[16].valid := 1, [565].log_data[17].valid := 1, [565].log_data[18].valid := 1, [565].log_data[19].valid := 1, [565].time.Year := 2023, [565].time.Month := 1, [565].time.Day := 13, [565].time.Hour := 13, [565].time.Minute := 44, [565].time.Second := 59, [566].log_data[0].min := 1.0, [566].log_data[0].max := 1.0, [566].log_data[0].total := 900.0, [566].log_data[0].time := 900.0, [566].log_data[0].minminute := 45, [566].log_data[0].maxminute := 45, [566].log_data[0].valid := 1, [566].log_data[1].valid := 1, [566].log_data[2].valid := 1, [566].log_data[3].valid := 1, [566].log_data[4].valid := 1, [566].log_data[5].valid := 1, [566].log_data[6].valid := 1, [566].log_data[7].valid := 1, [566].log_data[8].valid := 1, [566].log_data[9].valid := 1, [566].log_data[10].valid := 1, [566].log_data[11].valid := 1, [566].log_data[12].valid := 1,
        [566].log_data[13].valid := 1, [566].log_data[14].valid := 1, [566].log_data[15].valid := 1, [566].log_data[16].valid := 1, [566].log_data[17].valid := 1, [566].log_data[18].valid := 1, [566].log_data[19].valid := 1, [566].time.Year := 2023, [566].time.Month := 1, [566].time.Day := 13, [566].time.Hour := 13, [566].time.Minute := 59, [566].time.Second := 59, [567].log_data[0].min := 1.0, [567].log_data[0].max := 1.0, [567].log_data[0].total := 900.0, [567].log_data[0].time := 900.0, [567].log_data[0].valid := 1, [567].log_data[1].valid := 1, [567].log_data[2].valid := 1, [567].log_data[3].valid := 1, [567].log_data[4].valid := 1, [567].log_data[5].valid := 1, [567].log_data[6].valid := 1, [567].log_data[7].valid := 1, [567].log_data[8].valid := 1, [567].log_data[9].valid := 1, [567].log_data[10].valid := 1, [567].log_data[11].valid := 1, [567].log_data[12].valid := 1, [567].log_data[13].valid := 1, [567].log_data[14].valid := 1, [567].log_data[15].valid := 1, [567].log_data[16].valid := 1, [567].log_data[17].valid := 1, [567].log_data[18].valid := 1, [567].log_data[19].valid := 1, [567].time.Year := 2023, [567].time.Month := 1, [567].time.Day := 13, [567].time.Hour := 14, [567].time.Minute := 14, [567].time.Second := 59, [568].log_data[0].min := 1.0, [568].log_data[0].max := 1.0, [568].log_data[0].total := 900.0, [568].log_data[0].time := 900.0, [568].log_data[0].minminute := 15, [568].log_data[0].maxminute := 15, [568].log_data[0].valid := 1, [568].log_data[1].valid := 1, [568].log_data[2].valid := 1, [568].log_data[3].valid := 1, [568].log_data[4].valid := 1, [568].log_data[5].valid := 1, [568].log_data[6].valid := 1, [568].log_data[7].valid := 1, [568].log_data[8].valid := 1, [568].log_data[9].valid := 1, [568].log_data[10].valid := 1,
        [568].log_data[11].valid := 1, [568].log_data[12].valid := 1, [568].log_data[13].valid := 1, [568].log_data[14].valid := 1, [568].log_data[15].valid := 1, [568].log_data[16].valid := 1, [568].log_data[17].valid := 1, [568].log_data[18].valid := 1, [568].log_data[19].valid := 1, [568].time.Year := 2023, [568].time.Month := 1, [568].time.Day := 13, [568].time.Hour := 14, [568].time.Minute := 29, [568].time.Second := 59, [569].log_data[0].min := 1.0, [569].log_data[0].max := 1.0, [569].log_data[0].total := 900.0, [569].log_data[0].time := 900.0, [569].log_data[0].minminute := 30, [569].log_data[0].maxminute := 30, [569].log_data[0].valid := 1, [569].log_data[1].valid := 1, [569].log_data[2].valid := 1, [569].log_data[3].valid := 1, [569].log_data[4].valid := 1, [569].log_data[5].valid := 1, [569].log_data[6].valid := 1, [569].log_data[7].valid := 1, [569].log_data[8].valid := 1, [569].log_data[9].valid := 1, [569].log_data[10].valid := 1, [569].log_data[11].valid := 1, [569].log_data[12].valid := 1, [569].log_data[13].valid := 1, [569].log_data[14].valid := 1, [569].log_data[15].valid := 1, [569].log_data[16].valid := 1, [569].log_data[17].valid := 1, [569].log_data[18].valid := 1, [569].log_data[19].valid := 1, [569].time.Year := 2023, [569].time.Month := 1, [569].time.Day := 13, [569].time.Hour := 14, [569].time.Minute := 44, [569].time.Second := 59, [570].log_data[0].min := 1.0, [570].log_data[0].max := 1.0, [570].log_data[0].total := 900.0, [570].log_data[0].time := 900.0, [570].log_data[0].minminute := 45, [570].log_data[0].maxminute := 45, [570].log_data[0].valid := 1, [570].log_data[1].valid := 1, [570].log_data[2].valid := 1, [570].log_data[3].valid := 1, [570].log_data[4].valid := 1, [570].log_data[5].valid := 1, [570].log_data[6].valid := 1,
        [570].log_data[7].valid := 1, [570].log_data[8].valid := 1, [570].log_data[9].valid := 1, [570].log_data[10].valid := 1, [570].log_data[11].valid := 1, [570].log_data[12].valid := 1, [570].log_data[13].valid := 1, [570].log_data[14].valid := 1, [570].log_data[15].valid := 1, [570].log_data[16].valid := 1, [570].log_data[17].valid := 1, [570].log_data[18].valid := 1, [570].log_data[19].valid := 1, [570].time.Year := 2023, [570].time.Month := 1, [570].time.Day := 13, [570].time.Hour := 14, [570].time.Minute := 59, [570].time.Second := 59, [571].log_data[0].min := 1.0, [571].log_data[0].max := 1.0, [571].log_data[0].total := 900.0, [571].log_data[0].time := 900.0, [571].log_data[0].valid := 1, [571].log_data[1].valid := 1, [571].log_data[2].valid := 1, [571].log_data[3].valid := 1, [571].log_data[4].valid := 1, [571].log_data[5].valid := 1, [571].log_data[6].valid := 1, [571].log_data[7].valid := 1, [571].log_data[8].valid := 1, [571].log_data[9].valid := 1, [571].log_data[10].valid := 1, [571].log_data[11].valid := 1, [571].log_data[12].valid := 1, [571].log_data[13].valid := 1, [571].log_data[14].valid := 1, [571].log_data[15].valid := 1, [571].log_data[16].valid := 1, [571].log_data[17].valid := 1, [571].log_data[18].valid := 1, [571].log_data[19].valid := 1, [571].time.Year := 2023, [571].time.Month := 1, [571].time.Day := 13, [571].time.Hour := 15, [571].time.Minute := 14, [571].time.Second := 59, [572].log_data[0].min := 1.0, [572].log_data[0].max := 1.0, [572].log_data[0].total := 900.0, [572].log_data[0].time := 900.0, [572].log_data[0].minminute := 15, [572].log_data[0].maxminute := 15, [572].log_data[0].valid := 1, [572].log_data[1].valid := 1, [572].log_data[2].valid := 1, [572].log_data[3].valid := 1, [572].log_data[4].valid := 1,
        [572].log_data[5].valid := 1, [572].log_data[6].valid := 1, [572].log_data[7].valid := 1, [572].log_data[8].valid := 1, [572].log_data[9].valid := 1, [572].log_data[10].valid := 1, [572].log_data[11].valid := 1, [572].log_data[12].valid := 1, [572].log_data[13].valid := 1, [572].log_data[14].valid := 1, [572].log_data[15].valid := 1, [572].log_data[16].valid := 1, [572].log_data[17].valid := 1, [572].log_data[18].valid := 1, [572].log_data[19].valid := 1, [572].time.Year := 2023, [572].time.Month := 1, [572].time.Day := 13, [572].time.Hour := 15, [572].time.Minute := 29, [572].time.Second := 59, [573].log_data[0].min := 1.0, [573].log_data[0].max := 1.0, [573].log_data[0].total := 900.0, [573].log_data[0].time := 900.0, [573].log_data[0].minminute := 30, [573].log_data[0].maxminute := 30, [573].log_data[0].valid := 1, [573].log_data[1].valid := 1, [573].log_data[2].valid := 1, [573].log_data[3].valid := 1, [573].log_data[4].valid := 1, [573].log_data[5].valid := 1, [573].log_data[6].valid := 1, [573].log_data[7].valid := 1, [573].log_data[8].valid := 1, [573].log_data[9].valid := 1, [573].log_data[10].valid := 1, [573].log_data[11].valid := 1, [573].log_data[12].valid := 1, [573].log_data[13].valid := 1, [573].log_data[14].valid := 1, [573].log_data[15].valid := 1, [573].log_data[16].valid := 1, [573].log_data[17].valid := 1, [573].log_data[18].valid := 1, [573].log_data[19].valid := 1, [573].time.Year := 2023, [573].time.Month := 1, [573].time.Day := 13, [573].time.Hour := 15, [573].time.Minute := 44, [573].time.Second := 59, [574].log_data[0].min := 1.0, [574].log_data[0].max := 1.0, [574].log_data[0].total := 900.0, [574].log_data[0].time := 900.0, [574].log_data[0].minminute := 45, [574].log_data[0].maxminute := 45, [574].log_data[0].valid := 1,
        [574].log_data[1].valid := 1, [574].log_data[2].valid := 1, [574].log_data[3].valid := 1, [574].log_data[4].valid := 1, [574].log_data[5].valid := 1, [574].log_data[6].valid := 1, [574].log_data[7].valid := 1, [574].log_data[8].valid := 1, [574].log_data[9].valid := 1, [574].log_data[10].valid := 1, [574].log_data[11].valid := 1, [574].log_data[12].valid := 1, [574].log_data[13].valid := 1, [574].log_data[14].valid := 1, [574].log_data[15].valid := 1, [574].log_data[16].valid := 1, [574].log_data[17].valid := 1, [574].log_data[18].valid := 1, [574].log_data[19].valid := 1, [574].time.Year := 2023, [574].time.Month := 1, [574].time.Day := 13, [574].time.Hour := 15, [574].time.Minute := 59, [574].time.Second := 59, [575].log_data[0].min := 1.0, [575].log_data[0].max := 1.0, [575].log_data[0].total := 900.0, [575].log_data[0].time := 900.0, [575].log_data[0].valid := 1, [575].log_data[1].valid := 1, [575].log_data[2].valid := 1, [575].log_data[3].valid := 1, [575].log_data[4].valid := 1, [575].log_data[5].valid := 1, [575].log_data[6].valid := 1, [575].log_data[7].valid := 1, [575].log_data[8].valid := 1, [575].log_data[9].valid := 1, [575].log_data[10].valid := 1, [575].log_data[11].valid := 1, [575].log_data[12].valid := 1, [575].log_data[13].valid := 1, [575].log_data[14].valid := 1, [575].log_data[15].valid := 1, [575].log_data[16].valid := 1, [575].log_data[17].valid := 1, [575].log_data[18].valid := 1, [575].log_data[19].valid := 1, [575].time.Year := 2023, [575].time.Month := 1, [575].time.Day := 13, [575].time.Hour := 16, [575].time.Minute := 14, [575].time.Second := 59, [576].log_data[0].min := 1.0, [576].log_data[0].max := 1.0, [576].log_data[0].total := 900.0, [576].log_data[0].time := 900.0, [576].log_data[0].minminute := 15,
        [576].log_data[0].maxminute := 15, [576].log_data[0].valid := 1, [576].log_data[1].valid := 1, [576].log_data[2].valid := 1, [576].log_data[3].valid := 1, [576].log_data[4].valid := 1, [576].log_data[5].valid := 1, [576].log_data[6].valid := 1, [576].log_data[7].valid := 1, [576].log_data[8].valid := 1, [576].log_data[9].valid := 1, [576].log_data[10].valid := 1, [576].log_data[11].valid := 1, [576].log_data[12].valid := 1, [576].log_data[13].valid := 1, [576].log_data[14].valid := 1, [576].log_data[15].valid := 1, [576].log_data[16].valid := 1, [576].log_data[17].valid := 1, [576].log_data[18].valid := 1, [576].log_data[19].valid := 1, [576].time.Year := 2023, [576].time.Month := 1, [576].time.Day := 13, [576].time.Hour := 16, [576].time.Minute := 29, [576].time.Second := 59, [577].log_data[0].min := 1.0, [577].log_data[0].max := 1.0, [577].log_data[0].total := 900.0, [577].log_data[0].time := 900.0, [577].log_data[0].minminute := 30, [577].log_data[0].maxminute := 30, [577].log_data[0].valid := 1, [577].log_data[1].valid := 1, [577].log_data[2].valid := 1, [577].log_data[3].valid := 1, [577].log_data[4].valid := 1, [577].log_data[5].valid := 1, [577].log_data[6].valid := 1, [577].log_data[7].valid := 1, [577].log_data[8].valid := 1, [577].log_data[9].valid := 1, [577].log_data[10].valid := 1, [577].log_data[11].valid := 1, [577].log_data[12].valid := 1, [577].log_data[13].valid := 1, [577].log_data[14].valid := 1, [577].log_data[15].valid := 1, [577].log_data[16].valid := 1, [577].log_data[17].valid := 1, [577].log_data[18].valid := 1, [577].log_data[19].valid := 1, [577].time.Year := 2023, [577].time.Month := 1, [577].time.Day := 13, [577].time.Hour := 16, [577].time.Minute := 44, [577].time.Second := 59, [578].log_data[0].min := 1.0,
        [578].log_data[0].max := 1.0, [578].log_data[0].total := 900.0, [578].log_data[0].time := 900.0, [578].log_data[0].minminute := 45, [578].log_data[0].maxminute := 45, [578].log_data[0].valid := 1, [578].log_data[1].valid := 1, [578].log_data[2].valid := 1, [578].log_data[3].valid := 1, [578].log_data[4].valid := 1, [578].log_data[5].valid := 1, [578].log_data[6].valid := 1, [578].log_data[7].valid := 1, [578].log_data[8].valid := 1, [578].log_data[9].valid := 1, [578].log_data[10].valid := 1, [578].log_data[11].valid := 1, [578].log_data[12].valid := 1, [578].log_data[13].valid := 1, [578].log_data[14].valid := 1, [578].log_data[15].valid := 1, [578].log_data[16].valid := 1, [578].log_data[17].valid := 1, [578].log_data[18].valid := 1, [578].log_data[19].valid := 1, [578].time.Year := 2023, [578].time.Month := 1, [578].time.Day := 13, [578].time.Hour := 16, [578].time.Minute := 59, [578].time.Second := 59, [579].log_data[0].min := 1.0, [579].log_data[0].max := 1.0, [579].log_data[0].total := 900.0, [579].log_data[0].time := 900.0, [579].log_data[0].valid := 1, [579].log_data[1].valid := 1, [579].log_data[2].valid := 1, [579].log_data[3].valid := 1, [579].log_data[4].valid := 1, [579].log_data[5].valid := 1, [579].log_data[6].valid := 1, [579].log_data[7].valid := 1, [579].log_data[8].valid := 1, [579].log_data[9].valid := 1, [579].log_data[10].valid := 1, [579].log_data[11].valid := 1, [579].log_data[12].valid := 1, [579].log_data[13].valid := 1, [579].log_data[14].valid := 1, [579].log_data[15].valid := 1, [579].log_data[16].valid := 1, [579].log_data[17].valid := 1, [579].log_data[18].valid := 1, [579].log_data[19].valid := 1, [579].time.Year := 2023, [579].time.Month := 1, [579].time.Day := 13, [579].time.Hour := 17, [579].time.Minute := 14,
        [579].time.Second := 59, [580].log_data[0].min := 1.0, [580].log_data[0].max := 1.0, [580].log_data[0].total := 900.0, [580].log_data[0].time := 900.0, [580].log_data[0].minminute := 15, [580].log_data[0].maxminute := 15, [580].log_data[0].valid := 1, [580].log_data[1].valid := 1, [580].log_data[2].valid := 1, [580].log_data[3].valid := 1, [580].log_data[4].valid := 1, [580].log_data[5].valid := 1, [580].log_data[6].valid := 1, [580].log_data[7].valid := 1, [580].log_data[8].valid := 1, [580].log_data[9].valid := 1, [580].log_data[10].valid := 1, [580].log_data[11].valid := 1, [580].log_data[12].valid := 1, [580].log_data[13].valid := 1, [580].log_data[14].valid := 1, [580].log_data[15].valid := 1, [580].log_data[16].valid := 1, [580].log_data[17].valid := 1, [580].log_data[18].valid := 1, [580].log_data[19].valid := 1, [580].time.Year := 2023, [580].time.Month := 1, [580].time.Day := 13, [580].time.Hour := 17, [580].time.Minute := 29, [580].time.Second := 59, [581].log_data[0].min := 1.0, [581].log_data[0].max := 1.0, [581].log_data[0].total := 900.0, [581].log_data[0].time := 900.0, [581].log_data[0].minminute := 30, [581].log_data[0].maxminute := 30, [581].log_data[0].valid := 1, [581].log_data[1].valid := 1, [581].log_data[2].valid := 1, [581].log_data[3].valid := 1, [581].log_data[4].valid := 1, [581].log_data[5].valid := 1, [581].log_data[6].valid := 1, [581].log_data[7].valid := 1, [581].log_data[8].valid := 1, [581].log_data[9].valid := 1, [581].log_data[10].valid := 1, [581].log_data[11].valid := 1, [581].log_data[12].valid := 1, [581].log_data[13].valid := 1, [581].log_data[14].valid := 1, [581].log_data[15].valid := 1, [581].log_data[16].valid := 1, [581].log_data[17].valid := 1, [581].log_data[18].valid := 1, [581].log_data[19].valid := 1, [581].time.Year := 2023,
        [581].time.Month := 1, [581].time.Day := 13, [581].time.Hour := 17, [581].time.Minute := 44, [581].time.Second := 59, [582].log_data[0].min := 1.0, [582].log_data[0].max := 1.0, [582].log_data[0].total := 900.0, [582].log_data[0].time := 900.0, [582].log_data[0].minminute := 45, [582].log_data[0].maxminute := 45, [582].log_data[0].valid := 1, [582].log_data[1].valid := 1, [582].log_data[2].valid := 1, [582].log_data[3].valid := 1, [582].log_data[4].valid := 1, [582].log_data[5].valid := 1, [582].log_data[6].valid := 1, [582].log_data[7].valid := 1, [582].log_data[8].valid := 1, [582].log_data[9].valid := 1, [582].log_data[10].valid := 1, [582].log_data[11].valid := 1, [582].log_data[12].valid := 1, [582].log_data[13].valid := 1, [582].log_data[14].valid := 1, [582].log_data[15].valid := 1, [582].log_data[16].valid := 1, [582].log_data[17].valid := 1, [582].log_data[18].valid := 1, [582].log_data[19].valid := 1, [582].time.Year := 2023, [582].time.Month := 1, [582].time.Day := 13, [582].time.Hour := 17, [582].time.Minute := 59, [582].time.Second := 59, [583].log_data[0].min := 1.0, [583].log_data[0].max := 1.0, [583].log_data[0].total := 900.0, [583].log_data[0].time := 900.0, [583].log_data[0].valid := 1, [583].log_data[1].valid := 1, [583].log_data[2].valid := 1, [583].log_data[3].valid := 1, [583].log_data[4].valid := 1, [583].log_data[5].valid := 1, [583].log_data[6].valid := 1, [583].log_data[7].valid := 1, [583].log_data[8].valid := 1, [583].log_data[9].valid := 1, [583].log_data[10].valid := 1, [583].log_data[11].valid := 1, [583].log_data[12].valid := 1, [583].log_data[13].valid := 1, [583].log_data[14].valid := 1, [583].log_data[15].valid := 1, [583].log_data[16].valid := 1, [583].log_data[17].valid := 1, [583].log_data[18].valid := 1,
        [583].log_data[19].valid := 1, [583].time.Year := 2023, [583].time.Month := 1, [583].time.Day := 13, [583].time.Hour := 18, [583].time.Minute := 14, [583].time.Second := 59, [584].log_data[0].min := 1.0, [584].log_data[0].max := 1.0, [584].log_data[0].total := 900.0, [584].log_data[0].time := 900.0, [584].log_data[0].minminute := 15, [584].log_data[0].maxminute := 15, [584].log_data[0].valid := 1, [584].log_data[1].valid := 1, [584].log_data[2].valid := 1, [584].log_data[3].valid := 1, [584].log_data[4].valid := 1, [584].log_data[5].valid := 1, [584].log_data[6].valid := 1, [584].log_data[7].valid := 1, [584].log_data[8].valid := 1, [584].log_data[9].valid := 1, [584].log_data[10].valid := 1, [584].log_data[11].valid := 1, [584].log_data[12].valid := 1, [584].log_data[13].valid := 1, [584].log_data[14].valid := 1, [584].log_data[15].valid := 1, [584].log_data[16].valid := 1, [584].log_data[17].valid := 1, [584].log_data[18].valid := 1, [584].log_data[19].valid := 1, [584].time.Year := 2023, [584].time.Month := 1, [584].time.Day := 13, [584].time.Hour := 18, [584].time.Minute := 29, [584].time.Second := 59, [585].log_data[0].min := 1.0, [585].log_data[0].max := 1.0, [585].log_data[0].total := 900.0, [585].log_data[0].time := 900.0, [585].log_data[0].minminute := 30, [585].log_data[0].maxminute := 30, [585].log_data[0].valid := 1, [585].log_data[1].valid := 1, [585].log_data[2].valid := 1, [585].log_data[3].valid := 1, [585].log_data[4].valid := 1, [585].log_data[5].valid := 1, [585].log_data[6].valid := 1, [585].log_data[7].valid := 1, [585].log_data[8].valid := 1, [585].log_data[9].valid := 1, [585].log_data[10].valid := 1, [585].log_data[11].valid := 1, [585].log_data[12].valid := 1, [585].log_data[13].valid := 1, [585].log_data[14].valid := 1,
        [585].log_data[15].valid := 1, [585].log_data[16].valid := 1, [585].log_data[17].valid := 1, [585].log_data[18].valid := 1, [585].log_data[19].valid := 1, [585].time.Year := 2023, [585].time.Month := 1, [585].time.Day := 13, [585].time.Hour := 18, [585].time.Minute := 44, [585].time.Second := 59, [586].log_data[0].min := 1.0, [586].log_data[0].max := 1.0, [586].log_data[0].total := 900.0, [586].log_data[0].time := 900.0, [586].log_data[0].minminute := 45, [586].log_data[0].maxminute := 45, [586].log_data[0].valid := 1, [586].log_data[1].valid := 1, [586].log_data[2].valid := 1, [586].log_data[3].valid := 1, [586].log_data[4].valid := 1, [586].log_data[5].valid := 1, [586].log_data[6].valid := 1, [586].log_data[7].valid := 1, [586].log_data[8].valid := 1, [586].log_data[9].valid := 1, [586].log_data[10].valid := 1, [586].log_data[11].valid := 1, [586].log_data[12].valid := 1, [586].log_data[13].valid := 1, [586].log_data[14].valid := 1, [586].log_data[15].valid := 1, [586].log_data[16].valid := 1, [586].log_data[17].valid := 1, [586].log_data[18].valid := 1, [586].log_data[19].valid := 1, [586].time.Year := 2023, [586].time.Month := 1, [586].time.Day := 13, [586].time.Hour := 18, [586].time.Minute := 59, [586].time.Second := 59, [587].log_data[0].min := 1.0, [587].log_data[0].max := 1.0, [587].log_data[0].total := 900.0, [587].log_data[0].time := 900.0, [587].log_data[0].valid := 1, [587].log_data[1].valid := 1, [587].log_data[2].valid := 1, [587].log_data[3].valid := 1, [587].log_data[4].valid := 1, [587].log_data[5].valid := 1, [587].log_data[6].valid := 1, [587].log_data[7].valid := 1, [587].log_data[8].valid := 1, [587].log_data[9].valid := 1, [587].log_data[10].valid := 1, [587].log_data[11].valid := 1, [587].log_data[12].valid := 1,
        [587].log_data[13].valid := 1, [587].log_data[14].valid := 1, [587].log_data[15].valid := 1, [587].log_data[16].valid := 1, [587].log_data[17].valid := 1, [587].log_data[18].valid := 1, [587].log_data[19].valid := 1, [587].time.Year := 2023, [587].time.Month := 1, [587].time.Day := 13, [587].time.Hour := 19, [587].time.Minute := 14, [587].time.Second := 59, [588].log_data[0].min := 1.0, [588].log_data[0].max := 1.0, [588].log_data[0].total := 900.0, [588].log_data[0].time := 900.0, [588].log_data[0].minminute := 15, [588].log_data[0].maxminute := 15, [588].log_data[0].valid := 1, [588].log_data[1].valid := 1, [588].log_data[2].valid := 1, [588].log_data[3].valid := 1, [588].log_data[4].valid := 1, [588].log_data[5].valid := 1, [588].log_data[6].valid := 1, [588].log_data[7].valid := 1, [588].log_data[8].valid := 1, [588].log_data[9].valid := 1, [588].log_data[10].valid := 1, [588].log_data[11].valid := 1, [588].log_data[12].valid := 1, [588].log_data[13].valid := 1, [588].log_data[14].valid := 1, [588].log_data[15].valid := 1, [588].log_data[16].valid := 1, [588].log_data[17].valid := 1, [588].log_data[18].valid := 1, [588].log_data[19].valid := 1, [588].time.Year := 2023, [588].time.Month := 1, [588].time.Day := 13, [588].time.Hour := 19, [588].time.Minute := 29, [588].time.Second := 59, [589].log_data[0].min := 1.0, [589].log_data[0].max := 1.0, [589].log_data[0].total := 900.0, [589].log_data[0].time := 900.0, [589].log_data[0].minminute := 30, [589].log_data[0].maxminute := 30, [589].log_data[0].valid := 1, [589].log_data[1].valid := 1, [589].log_data[2].valid := 1, [589].log_data[3].valid := 1, [589].log_data[4].valid := 1, [589].log_data[5].valid := 1, [589].log_data[6].valid := 1, [589].log_data[7].valid := 1, [589].log_data[8].valid := 1,
        [589].log_data[9].valid := 1, [589].log_data[10].valid := 1, [589].log_data[11].valid := 1, [589].log_data[12].valid := 1, [589].log_data[13].valid := 1, [589].log_data[14].valid := 1, [589].log_data[15].valid := 1, [589].log_data[16].valid := 1, [589].log_data[17].valid := 1, [589].log_data[18].valid := 1, [589].log_data[19].valid := 1, [589].time.Year := 2023, [589].time.Month := 1, [589].time.Day := 13, [589].time.Hour := 19, [589].time.Minute := 44, [589].time.Second := 59, [590].log_data[0].min := 1.0, [590].log_data[0].max := 1.0, [590].log_data[0].total := 900.0, [590].log_data[0].time := 900.0, [590].log_data[0].minminute := 45, [590].log_data[0].maxminute := 45, [590].log_data[0].valid := 1, [590].log_data[1].valid := 1, [590].log_data[2].valid := 1, [590].log_data[3].valid := 1, [590].log_data[4].valid := 1, [590].log_data[5].valid := 1, [590].log_data[6].valid := 1, [590].log_data[7].valid := 1, [590].log_data[8].valid := 1, [590].log_data[9].valid := 1, [590].log_data[10].valid := 1, [590].log_data[11].valid := 1, [590].log_data[12].valid := 1, [590].log_data[13].valid := 1, [590].log_data[14].valid := 1, [590].log_data[15].valid := 1, [590].log_data[16].valid := 1, [590].log_data[17].valid := 1, [590].log_data[18].valid := 1, [590].log_data[19].valid := 1, [590].time.Year := 2023, [590].time.Month := 1, [590].time.Day := 13, [590].time.Hour := 19, [590].time.Minute := 59, [590].time.Second := 59, [591].log_data[0].min := 1.0, [591].log_data[0].max := 1.0, [591].log_data[0].total := 900.0, [591].log_data[0].time := 900.0, [591].log_data[0].valid := 1, [591].log_data[1].valid := 1, [591].log_data[2].valid := 1, [591].log_data[3].valid := 1, [591].log_data[4].valid := 1, [591].log_data[5].valid := 1, [591].log_data[6].valid := 1,
        [591].log_data[7].valid := 1, [591].log_data[8].valid := 1, [591].log_data[9].valid := 1, [591].log_data[10].valid := 1, [591].log_data[11].valid := 1, [591].log_data[12].valid := 1, [591].log_data[13].valid := 1, [591].log_data[14].valid := 1, [591].log_data[15].valid := 1, [591].log_data[16].valid := 1, [591].log_data[17].valid := 1, [591].log_data[18].valid := 1, [591].log_data[19].valid := 1, [591].time.Year := 2023, [591].time.Month := 1, [591].time.Day := 13, [591].time.Hour := 20, [591].time.Minute := 14, [591].time.Second := 59, [592].log_data[0].min := 1.0, [592].log_data[0].max := 1.0, [592].log_data[0].total := 900.0, [592].log_data[0].time := 900.0, [592].log_data[0].minminute := 15, [592].log_data[0].maxminute := 15, [592].log_data[0].valid := 1, [592].log_data[1].valid := 1, [592].log_data[2].valid := 1, [592].log_data[3].valid := 1, [592].log_data[4].valid := 1, [592].log_data[5].valid := 1, [592].log_data[6].valid := 1, [592].log_data[7].valid := 1, [592].log_data[8].valid := 1, [592].log_data[9].valid := 1, [592].log_data[10].valid := 1, [592].log_data[11].valid := 1, [592].log_data[12].valid := 1, [592].log_data[13].valid := 1, [592].log_data[14].valid := 1, [592].log_data[15].valid := 1, [592].log_data[16].valid := 1, [592].log_data[17].valid := 1, [592].log_data[18].valid := 1, [592].log_data[19].valid := 1, [592].time.Year := 2023, [592].time.Month := 1, [592].time.Day := 13, [592].time.Hour := 20, [592].time.Minute := 29, [592].time.Second := 59, [593].log_data[0].min := 1.0, [593].log_data[0].max := 1.0, [593].log_data[0].total := 900.0, [593].log_data[0].time := 900.0, [593].log_data[0].minminute := 30, [593].log_data[0].maxminute := 30, [593].log_data[0].valid := 1, [593].log_data[1].valid := 1, [593].log_data[2].valid := 1,
        [593].log_data[3].valid := 1, [593].log_data[4].valid := 1, [593].log_data[5].valid := 1, [593].log_data[6].valid := 1, [593].log_data[7].valid := 1, [593].log_data[8].valid := 1, [593].log_data[9].valid := 1, [593].log_data[10].valid := 1, [593].log_data[11].valid := 1, [593].log_data[12].valid := 1, [593].log_data[13].valid := 1, [593].log_data[14].valid := 1, [593].log_data[15].valid := 1, [593].log_data[16].valid := 1, [593].log_data[17].valid := 1, [593].log_data[18].valid := 1, [593].log_data[19].valid := 1, [593].time.Year := 2023, [593].time.Month := 1, [593].time.Day := 13, [593].time.Hour := 20, [593].time.Minute := 44, [593].time.Second := 59, [594].log_data[0].min := 1.0, [594].log_data[0].max := 1.0, [594].log_data[0].total := 900.0, [594].log_data[0].time := 900.0, [594].log_data[0].minminute := 45, [594].log_data[0].maxminute := 45, [594].log_data[0].valid := 1, [594].log_data[1].valid := 1, [594].log_data[2].valid := 1, [594].log_data[3].valid := 1, [594].log_data[4].valid := 1, [594].log_data[5].valid := 1, [594].log_data[6].valid := 1, [594].log_data[7].valid := 1, [594].log_data[8].valid := 1, [594].log_data[9].valid := 1, [594].log_data[10].valid := 1, [594].log_data[11].valid := 1, [594].log_data[12].valid := 1, [594].log_data[13].valid := 1, [594].log_data[14].valid := 1, [594].log_data[15].valid := 1, [594].log_data[16].valid := 1, [594].log_data[17].valid := 1, [594].log_data[18].valid := 1, [594].log_data[19].valid := 1, [594].time.Year := 2023, [594].time.Month := 1, [594].time.Day := 13, [594].time.Hour := 20, [594].time.Minute := 59, [594].time.Second := 59, [595].log_data[0].min := 1.0, [595].log_data[0].max := 1.0, [595].log_data[0].total := 900.0, [595].log_data[0].time := 900.0, [595].log_data[0].valid := 1,
        [595].log_data[1].valid := 1, [595].log_data[2].valid := 1, [595].log_data[3].valid := 1, [595].log_data[4].valid := 1, [595].log_data[5].valid := 1, [595].log_data[6].valid := 1, [595].log_data[7].valid := 1, [595].log_data[8].valid := 1, [595].log_data[9].valid := 1, [595].log_data[10].valid := 1, [595].log_data[11].valid := 1, [595].log_data[12].valid := 1, [595].log_data[13].valid := 1, [595].log_data[14].valid := 1, [595].log_data[15].valid := 1, [595].log_data[16].valid := 1, [595].log_data[17].valid := 1, [595].log_data[18].valid := 1, [595].log_data[19].valid := 1, [595].time.Year := 2023, [595].time.Month := 1, [595].time.Day := 13, [595].time.Hour := 21, [595].time.Minute := 14, [595].time.Second := 59, [596].log_data[0].min := 1.0, [596].log_data[0].max := 1.0, [596].log_data[0].total := 900.0, [596].log_data[0].time := 900.0, [596].log_data[0].minminute := 15, [596].log_data[0].maxminute := 15, [596].log_data[0].valid := 1, [596].log_data[1].valid := 1, [596].log_data[2].valid := 1, [596].log_data[3].valid := 1, [596].log_data[4].valid := 1, [596].log_data[5].valid := 1, [596].log_data[6].valid := 1, [596].log_data[7].valid := 1, [596].log_data[8].valid := 1, [596].log_data[9].valid := 1, [596].log_data[10].valid := 1, [596].log_data[11].valid := 1, [596].log_data[12].valid := 1, [596].log_data[13].valid := 1, [596].log_data[14].valid := 1, [596].log_data[15].valid := 1, [596].log_data[16].valid := 1, [596].log_data[17].valid := 1, [596].log_data[18].valid := 1, [596].log_data[19].valid := 1, [596].time.Year := 2023, [596].time.Month := 1, [596].time.Day := 13, [596].time.Hour := 21, [596].time.Minute := 29, [596].time.Second := 59, [597].log_data[0].min := 1.0, [597].log_data[0].max := 1.0, [597].log_data[0].total := 900.0,
        [597].log_data[0].time := 900.0, [597].log_data[0].minminute := 30, [597].log_data[0].maxminute := 30, [597].log_data[0].valid := 1, [597].log_data[1].valid := 1, [597].log_data[2].valid := 1, [597].log_data[3].valid := 1, [597].log_data[4].valid := 1, [597].log_data[5].valid := 1, [597].log_data[6].valid := 1, [597].log_data[7].valid := 1, [597].log_data[8].valid := 1, [597].log_data[9].valid := 1, [597].log_data[10].valid := 1, [597].log_data[11].valid := 1, [597].log_data[12].valid := 1, [597].log_data[13].valid := 1, [597].log_data[14].valid := 1, [597].log_data[15].valid := 1, [597].log_data[16].valid := 1, [597].log_data[17].valid := 1, [597].log_data[18].valid := 1, [597].log_data[19].valid := 1, [597].time.Year := 2023, [597].time.Month := 1, [597].time.Day := 13, [597].time.Hour := 21, [597].time.Minute := 44, [597].time.Second := 59, [598].log_data[0].min := 1.0, [598].log_data[0].max := 1.0, [598].log_data[0].total := 900.0, [598].log_data[0].time := 900.0, [598].log_data[0].minminute := 45, [598].log_data[0].maxminute := 45, [598].log_data[0].valid := 1, [598].log_data[1].valid := 1, [598].log_data[2].valid := 1, [598].log_data[3].valid := 1, [598].log_data[4].valid := 1, [598].log_data[5].valid := 1, [598].log_data[6].valid := 1, [598].log_data[7].valid := 1, [598].log_data[8].valid := 1, [598].log_data[9].valid := 1, [598].log_data[10].valid := 1, [598].log_data[11].valid := 1, [598].log_data[12].valid := 1, [598].log_data[13].valid := 1, [598].log_data[14].valid := 1, [598].log_data[15].valid := 1, [598].log_data[16].valid := 1, [598].log_data[17].valid := 1, [598].log_data[18].valid := 1, [598].log_data[19].valid := 1, [598].time.Year := 2023, [598].time.Month := 1, [598].time.Day := 13, [598].time.Hour := 21, [598].time.Minute := 59,
        [598].time.Second := 59, [599].log_data[0].min := 1.0, [599].log_data[0].max := 1.0, [599].log_data[0].total := 900.0, [599].log_data[0].time := 900.0, [599].log_data[0].valid := 1, [599].log_data[1].valid := 1, [599].log_data[2].valid := 1, [599].log_data[3].valid := 1, [599].log_data[4].valid := 1, [599].log_data[5].valid := 1, [599].log_data[6].valid := 1, [599].log_data[7].valid := 1, [599].log_data[8].valid := 1, [599].log_data[9].valid := 1, [599].log_data[10].valid := 1, [599].log_data[11].valid := 1, [599].log_data[12].valid := 1, [599].log_data[13].valid := 1, [599].log_data[14].valid := 1, [599].log_data[15].valid := 1, [599].log_data[16].valid := 1, [599].log_data[17].valid := 1, [599].log_data[18].valid := 1, [599].log_data[19].valid := 1, [599].time.Year := 2023, [599].time.Month := 1, [599].time.Day := 13, [599].time.Hour := 22, [599].time.Minute := 14, [599].time.Second := 59, [600].log_data[0].min := 1.0, [600].log_data[0].max := 1.0, [600].log_data[0].total := 900.0, [600].log_data[0].time := 900.0, [600].log_data[0].minminute := 15, [600].log_data[0].maxminute := 15, [600].log_data[0].valid := 1, [600].log_data[1].valid := 1, [600].log_data[2].valid := 1, [600].log_data[3].valid := 1, [600].log_data[4].valid := 1, [600].log_data[5].valid := 1, [600].log_data[6].valid := 1, [600].log_data[7].valid := 1, [600].log_data[8].valid := 1, [600].log_data[9].valid := 1, [600].log_data[10].valid := 1, [600].log_data[11].valid := 1, [600].log_data[12].valid := 1, [600].log_data[13].valid := 1, [600].log_data[14].valid := 1, [600].log_data[15].valid := 1, [600].log_data[16].valid := 1, [600].log_data[17].valid := 1, [600].log_data[18].valid := 1, [600].log_data[19].valid := 1, [600].time.Year := 2023, [600].time.Month := 1, [600].time.Day := 13,
        [600].time.Hour := 22, [600].time.Minute := 29, [600].time.Second := 59, [601].log_data[0].min := 1.0, [601].log_data[0].max := 1.0, [601].log_data[0].total := 900.0, [601].log_data[0].time := 900.0, [601].log_data[0].minminute := 30, [601].log_data[0].maxminute := 30, [601].log_data[0].valid := 1, [601].log_data[1].valid := 1, [601].log_data[2].valid := 1, [601].log_data[3].valid := 1, [601].log_data[4].valid := 1, [601].log_data[5].valid := 1, [601].log_data[6].valid := 1, [601].log_data[7].valid := 1, [601].log_data[8].valid := 1, [601].log_data[9].valid := 1, [601].log_data[10].valid := 1, [601].log_data[11].valid := 1, [601].log_data[12].valid := 1, [601].log_data[13].valid := 1, [601].log_data[14].valid := 1, [601].log_data[15].valid := 1, [601].log_data[16].valid := 1, [601].log_data[17].valid := 1, [601].log_data[18].valid := 1, [601].log_data[19].valid := 1, [601].time.Year := 2023, [601].time.Month := 1, [601].time.Day := 13, [601].time.Hour := 22, [601].time.Minute := 44, [601].time.Second := 59, [602].log_data[0].min := 1.0, [602].log_data[0].max := 1.0, [602].log_data[0].total := 900.0, [602].log_data[0].time := 900.0, [602].log_data[0].minminute := 45, [602].log_data[0].maxminute := 45, [602].log_data[0].valid := 1, [602].log_data[1].valid := 1, [602].log_data[2].valid := 1, [602].log_data[3].valid := 1, [602].log_data[4].valid := 1, [602].log_data[5].valid := 1, [602].log_data[6].valid := 1, [602].log_data[7].valid := 1, [602].log_data[8].valid := 1, [602].log_data[9].valid := 1, [602].log_data[10].valid := 1, [602].log_data[11].valid := 1, [602].log_data[12].valid := 1, [602].log_data[13].valid := 1, [602].log_data[14].valid := 1, [602].log_data[15].valid := 1, [602].log_data[16].valid := 1, [602].log_data[17].valid := 1, [602].log_data[18].valid := 1,
        [602].log_data[19].valid := 1, [602].time.Year := 2023, [602].time.Month := 1, [602].time.Day := 13, [602].time.Hour := 22, [602].time.Minute := 59, [602].time.Second := 59, [603].log_data[0].min := 1.0, [603].log_data[0].max := 1.0, [603].log_data[0].total := 900.0, [603].log_data[0].time := 900.0, [603].log_data[0].valid := 1, [603].log_data[1].valid := 1, [603].log_data[2].valid := 1, [603].log_data[3].valid := 1, [603].log_data[4].valid := 1, [603].log_data[5].valid := 1, [603].log_data[6].valid := 1, [603].log_data[7].valid := 1, [603].log_data[8].valid := 1, [603].log_data[9].valid := 1, [603].log_data[10].valid := 1, [603].log_data[11].valid := 1, [603].log_data[12].valid := 1, [603].log_data[13].valid := 1, [603].log_data[14].valid := 1, [603].log_data[15].valid := 1, [603].log_data[16].valid := 1, [603].log_data[17].valid := 1, [603].log_data[18].valid := 1, [603].log_data[19].valid := 1, [603].time.Year := 2023, [603].time.Month := 1, [603].time.Day := 13, [603].time.Hour := 23, [603].time.Minute := 14, [603].time.Second := 59, [604].log_data[0].min := 1.0, [604].log_data[0].max := 1.0, [604].log_data[0].total := 900.0, [604].log_data[0].time := 900.0, [604].log_data[0].minminute := 15, [604].log_data[0].maxminute := 15, [604].log_data[0].valid := 1, [604].log_data[1].valid := 1, [604].log_data[2].valid := 1, [604].log_data[3].valid := 1, [604].log_data[4].valid := 1, [604].log_data[5].valid := 1, [604].log_data[6].valid := 1, [604].log_data[7].valid := 1, [604].log_data[8].valid := 1, [604].log_data[9].valid := 1, [604].log_data[10].valid := 1, [604].log_data[11].valid := 1, [604].log_data[12].valid := 1, [604].log_data[13].valid := 1, [604].log_data[14].valid := 1, [604].log_data[15].valid := 1, [604].log_data[16].valid := 1,
        [604].log_data[17].valid := 1, [604].log_data[18].valid := 1, [604].log_data[19].valid := 1, [604].time.Year := 2023, [604].time.Month := 1, [604].time.Day := 13, [604].time.Hour := 23, [604].time.Minute := 29, [604].time.Second := 59, [605].log_data[0].min := 1.0, [605].log_data[0].max := 1.0, [605].log_data[0].total := 900.0, [605].log_data[0].time := 900.0, [605].log_data[0].minminute := 30, [605].log_data[0].maxminute := 30, [605].log_data[0].valid := 1, [605].log_data[1].valid := 1, [605].log_data[2].valid := 1, [605].log_data[3].valid := 1, [605].log_data[4].valid := 1, [605].log_data[5].valid := 1, [605].log_data[6].valid := 1, [605].log_data[7].valid := 1, [605].log_data[8].valid := 1, [605].log_data[9].valid := 1, [605].log_data[10].valid := 1, [605].log_data[11].valid := 1, [605].log_data[12].valid := 1, [605].log_data[13].valid := 1, [605].log_data[14].valid := 1, [605].log_data[15].valid := 1, [605].log_data[16].valid := 1, [605].log_data[17].valid := 1, [605].log_data[18].valid := 1, [605].log_data[19].valid := 1, [605].time.Year := 2023, [605].time.Month := 1, [605].time.Day := 13, [605].time.Hour := 23, [605].time.Minute := 44, [605].time.Second := 59, [606].log_data[0].min := 1.0, [606].log_data[0].max := 1.0, [606].log_data[0].total := 900.0, [606].log_data[0].time := 900.0, [606].log_data[0].minminute := 45, [606].log_data[0].maxminute := 45, [606].log_data[0].valid := 1, [606].log_data[1].valid := 1, [606].log_data[2].valid := 1, [606].log_data[3].valid := 1, [606].log_data[4].valid := 1, [606].log_data[5].valid := 1, [606].log_data[6].valid := 1, [606].log_data[7].valid := 1, [606].log_data[8].valid := 1, [606].log_data[9].valid := 1, [606].log_data[10].valid := 1, [606].log_data[11].valid := 1, [606].log_data[12].valid := 1,
        [606].log_data[13].valid := 1, [606].log_data[14].valid := 1, [606].log_data[15].valid := 1, [606].log_data[16].valid := 1, [606].log_data[17].valid := 1, [606].log_data[18].valid := 1, [606].log_data[19].valid := 1, [606].time.Year := 2023, [606].time.Month := 1, [606].time.Day := 13, [606].time.Hour := 23, [606].time.Minute := 59, [606].time.Second := 59, [607].log_data[0].min := 1.0, [607].log_data[0].max := 1.0, [607].log_data[0].total := 899.5, [607].log_data[0].time := 899.5, [607].log_data[0].valid := 1, [607].log_data[1].valid := 1, [607].log_data[2].valid := 1, [607].log_data[3].valid := 1, [607].log_data[4].valid := 1, [607].log_data[5].valid := 1, [607].log_data[6].valid := 1, [607].log_data[7].valid := 1, [607].log_data[8].valid := 1, [607].log_data[9].valid := 1, [607].log_data[10].valid := 1, [607].log_data[11].valid := 1, [607].log_data[12].valid := 1, [607].log_data[13].valid := 1, [607].log_data[14].valid := 1, [607].log_data[15].valid := 1, [607].log_data[16].valid := 1, [607].log_data[17].valid := 1, [607].log_data[18].valid := 1, [607].log_data[19].valid := 1, [607].time.Year := 2023, [607].time.Month := 1, [607].time.Day := 14, [607].time.Minute := 14, [607].time.Second := 59, [608].log_data[0].min := 1.0, [608].log_data[0].max := 1.0, [608].log_data[0].total := 900.0, [608].log_data[0].time := 900.0, [608].log_data[0].minminute := 15, [608].log_data[0].maxminute := 15, [608].log_data[0].valid := 1, [608].log_data[1].valid := 1, [608].log_data[2].valid := 1, [608].log_data[3].valid := 1, [608].log_data[4].valid := 1, [608].log_data[5].valid := 1, [608].log_data[6].valid := 1, [608].log_data[7].valid := 1, [608].log_data[8].valid := 1, [608].log_data[9].valid := 1, [608].log_data[10].valid := 1, [608].log_data[11].valid := 1,
        [608].log_data[12].valid := 1, [608].log_data[13].valid := 1, [608].log_data[14].valid := 1, [608].log_data[15].valid := 1, [608].log_data[16].valid := 1, [608].log_data[17].valid := 1, [608].log_data[18].valid := 1, [608].log_data[19].valid := 1, [608].time.Year := 2023, [608].time.Month := 1, [608].time.Day := 14, [608].time.Minute := 29, [608].time.Second := 59, [609].log_data[0].min := 1.0, [609].log_data[0].max := 1.0, [609].log_data[0].total := 900.0, [609].log_data[0].time := 900.0, [609].log_data[0].minminute := 30, [609].log_data[0].maxminute := 30, [609].log_data[0].valid := 1, [609].log_data[1].valid := 1, [609].log_data[2].valid := 1, [609].log_data[3].valid := 1, [609].log_data[4].valid := 1, [609].log_data[5].valid := 1, [609].log_data[6].valid := 1, [609].log_data[7].valid := 1, [609].log_data[8].valid := 1, [609].log_data[9].valid := 1, [609].log_data[10].valid := 1, [609].log_data[11].valid := 1, [609].log_data[12].valid := 1, [609].log_data[13].valid := 1, [609].log_data[14].valid := 1, [609].log_data[15].valid := 1, [609].log_data[16].valid := 1, [609].log_data[17].valid := 1, [609].log_data[18].valid := 1, [609].log_data[19].valid := 1, [609].time.Year := 2023, [609].time.Month := 1, [609].time.Day := 14, [609].time.Minute := 44, [609].time.Second := 59, [610].log_data[0].min := 1.0, [610].log_data[0].max := 1.0, [610].log_data[0].total := 900.0, [610].log_data[0].time := 900.0, [610].log_data[0].minminute := 45, [610].log_data[0].maxminute := 45, [610].log_data[0].valid := 1, [610].log_data[1].valid := 1, [610].log_data[2].valid := 1, [610].log_data[3].valid := 1, [610].log_data[4].valid := 1, [610].log_data[5].valid := 1, [610].log_data[6].valid := 1, [610].log_data[7].valid := 1, [610].log_data[8].valid := 1, [610].log_data[9].valid := 1,
        [610].log_data[10].valid := 1, [610].log_data[11].valid := 1, [610].log_data[12].valid := 1, [610].log_data[13].valid := 1, [610].log_data[14].valid := 1, [610].log_data[15].valid := 1, [610].log_data[16].valid := 1, [610].log_data[17].valid := 1, [610].log_data[18].valid := 1, [610].log_data[19].valid := 1, [610].time.Year := 2023, [610].time.Month := 1, [610].time.Day := 14, [610].time.Minute := 59, [610].time.Second := 59, [611].log_data[0].min := 1.0, [611].log_data[0].max := 1.0, [611].log_data[0].total := 900.0, [611].log_data[0].time := 900.0, [611].log_data[0].valid := 1, [611].log_data[1].valid := 1, [611].log_data[2].valid := 1, [611].log_data[3].valid := 1, [611].log_data[4].valid := 1, [611].log_data[5].valid := 1, [611].log_data[6].valid := 1, [611].log_data[7].valid := 1, [611].log_data[8].valid := 1, [611].log_data[9].valid := 1, [611].log_data[10].valid := 1, [611].log_data[11].valid := 1, [611].log_data[12].valid := 1, [611].log_data[13].valid := 1, [611].log_data[14].valid := 1, [611].log_data[15].valid := 1, [611].log_data[16].valid := 1, [611].log_data[17].valid := 1, [611].log_data[18].valid := 1, [611].log_data[19].valid := 1, [611].time.Year := 2023, [611].time.Month := 1, [611].time.Day := 14, [611].time.Hour := 1, [611].time.Minute := 14, [611].time.Second := 59, [612].log_data[0].min := 1.0, [612].log_data[0].max := 1.0, [612].log_data[0].total := 900.0, [612].log_data[0].time := 900.0, [612].log_data[0].minminute := 15, [612].log_data[0].maxminute := 15, [612].log_data[0].valid := 1, [612].log_data[1].valid := 1, [612].log_data[2].valid := 1, [612].log_data[3].valid := 1, [612].log_data[4].valid := 1, [612].log_data[5].valid := 1, [612].log_data[6].valid := 1, [612].log_data[7].valid := 1, [612].log_data[8].valid := 1,
        [612].log_data[9].valid := 1, [612].log_data[10].valid := 1, [612].log_data[11].valid := 1, [612].log_data[12].valid := 1, [612].log_data[13].valid := 1, [612].log_data[14].valid := 1, [612].log_data[15].valid := 1, [612].log_data[16].valid := 1, [612].log_data[17].valid := 1, [612].log_data[18].valid := 1, [612].log_data[19].valid := 1, [612].time.Year := 2023, [612].time.Month := 1, [612].time.Day := 14, [612].time.Hour := 1, [612].time.Minute := 29, [612].time.Second := 59, [613].log_data[0].min := 1.0, [613].log_data[0].max := 1.0, [613].log_data[0].total := 900.0, [613].log_data[0].time := 900.0, [613].log_data[0].minminute := 30, [613].log_data[0].maxminute := 30, [613].log_data[0].valid := 1, [613].log_data[1].valid := 1, [613].log_data[2].valid := 1, [613].log_data[3].valid := 1, [613].log_data[4].valid := 1, [613].log_data[5].valid := 1, [613].log_data[6].valid := 1, [613].log_data[7].valid := 1, [613].log_data[8].valid := 1, [613].log_data[9].valid := 1, [613].log_data[10].valid := 1, [613].log_data[11].valid := 1, [613].log_data[12].valid := 1, [613].log_data[13].valid := 1, [613].log_data[14].valid := 1, [613].log_data[15].valid := 1, [613].log_data[16].valid := 1, [613].log_data[17].valid := 1, [613].log_data[18].valid := 1, [613].log_data[19].valid := 1, [613].time.Year := 2023, [613].time.Month := 1, [613].time.Day := 14, [613].time.Hour := 1, [613].time.Minute := 44, [613].time.Second := 59, [614].log_data[0].min := 1.0, [614].log_data[0].max := 1.0, [614].log_data[0].total := 900.0, [614].log_data[0].time := 900.0, [614].log_data[0].minminute := 45, [614].log_data[0].maxminute := 45, [614].log_data[0].valid := 1, [614].log_data[1].valid := 1, [614].log_data[2].valid := 1, [614].log_data[3].valid := 1, [614].log_data[4].valid := 1,
        [614].log_data[5].valid := 1, [614].log_data[6].valid := 1, [614].log_data[7].valid := 1, [614].log_data[8].valid := 1, [614].log_data[9].valid := 1, [614].log_data[10].valid := 1, [614].log_data[11].valid := 1, [614].log_data[12].valid := 1, [614].log_data[13].valid := 1, [614].log_data[14].valid := 1, [614].log_data[15].valid := 1, [614].log_data[16].valid := 1, [614].log_data[17].valid := 1, [614].log_data[18].valid := 1, [614].log_data[19].valid := 1, [614].time.Year := 2023, [614].time.Month := 1, [614].time.Day := 14, [614].time.Hour := 1, [614].time.Minute := 59, [614].time.Second := 59, [615].log_data[0].min := 1.0, [615].log_data[0].max := 1.0, [615].log_data[0].total := 900.0, [615].log_data[0].time := 900.0, [615].log_data[0].valid := 1, [615].log_data[1].valid := 1, [615].log_data[2].valid := 1, [615].log_data[3].valid := 1, [615].log_data[4].valid := 1, [615].log_data[5].valid := 1, [615].log_data[6].valid := 1, [615].log_data[7].valid := 1, [615].log_data[8].valid := 1, [615].log_data[9].valid := 1, [615].log_data[10].valid := 1, [615].log_data[11].valid := 1, [615].log_data[12].valid := 1, [615].log_data[13].valid := 1, [615].log_data[14].valid := 1, [615].log_data[15].valid := 1, [615].log_data[16].valid := 1, [615].log_data[17].valid := 1, [615].log_data[18].valid := 1, [615].log_data[19].valid := 1, [615].time.Year := 2023, [615].time.Month := 1, [615].time.Day := 14, [615].time.Hour := 2, [615].time.Minute := 14, [615].time.Second := 59, [616].log_data[0].min := 1.0, [616].log_data[0].max := 1.0, [616].log_data[0].total := 900.0, [616].log_data[0].time := 900.0, [616].log_data[0].minminute := 15, [616].log_data[0].maxminute := 15, [616].log_data[0].valid := 1, [616].log_data[1].valid := 1, [616].log_data[2].valid := 1,
        [616].log_data[3].valid := 1, [616].log_data[4].valid := 1, [616].log_data[5].valid := 1, [616].log_data[6].valid := 1, [616].log_data[7].valid := 1, [616].log_data[8].valid := 1, [616].log_data[9].valid := 1, [616].log_data[10].valid := 1, [616].log_data[11].valid := 1, [616].log_data[12].valid := 1, [616].log_data[13].valid := 1, [616].log_data[14].valid := 1, [616].log_data[15].valid := 1, [616].log_data[16].valid := 1, [616].log_data[17].valid := 1, [616].log_data[18].valid := 1, [616].log_data[19].valid := 1, [616].time.Year := 2023, [616].time.Month := 1, [616].time.Day := 14, [616].time.Hour := 2, [616].time.Minute := 29, [616].time.Second := 59, [617].log_data[0].min := 1.0, [617].log_data[0].max := 1.0, [617].log_data[0].total := 900.0, [617].log_data[0].time := 900.0, [617].log_data[0].minminute := 30, [617].log_data[0].maxminute := 30, [617].log_data[0].valid := 1, [617].log_data[1].valid := 1, [617].log_data[2].valid := 1, [617].log_data[3].valid := 1, [617].log_data[4].valid := 1, [617].log_data[5].valid := 1, [617].log_data[6].valid := 1, [617].log_data[7].valid := 1, [617].log_data[8].valid := 1, [617].log_data[9].valid := 1, [617].log_data[10].valid := 1, [617].log_data[11].valid := 1, [617].log_data[12].valid := 1, [617].log_data[13].valid := 1, [617].log_data[14].valid := 1, [617].log_data[15].valid := 1, [617].log_data[16].valid := 1, [617].log_data[17].valid := 1, [617].log_data[18].valid := 1, [617].log_data[19].valid := 1, [617].time.Year := 2023, [617].time.Month := 1, [617].time.Day := 14, [617].time.Hour := 2, [617].time.Minute := 44, [617].time.Second := 59, [618].log_data[0].min := 1.0, [618].log_data[0].max := 1.0, [618].log_data[0].total := 900.0, [618].log_data[0].time := 900.0, [618].log_data[0].minminute := 45,
        [618].log_data[0].maxminute := 45, [618].log_data[0].valid := 1, [618].log_data[1].valid := 1, [618].log_data[2].valid := 1, [618].log_data[3].valid := 1, [618].log_data[4].valid := 1, [618].log_data[5].valid := 1, [618].log_data[6].valid := 1, [618].log_data[7].valid := 1, [618].log_data[8].valid := 1, [618].log_data[9].valid := 1, [618].log_data[10].valid := 1, [618].log_data[11].valid := 1, [618].log_data[12].valid := 1, [618].log_data[13].valid := 1, [618].log_data[14].valid := 1, [618].log_data[15].valid := 1, [618].log_data[16].valid := 1, [618].log_data[17].valid := 1, [618].log_data[18].valid := 1, [618].log_data[19].valid := 1, [618].time.Year := 2023, [618].time.Month := 1, [618].time.Day := 14, [618].time.Hour := 2, [618].time.Minute := 59, [618].time.Second := 59, [619].log_data[0].min := 1.0, [619].log_data[0].max := 1.0, [619].log_data[0].total := 900.0, [619].log_data[0].time := 900.0, [619].log_data[0].valid := 1, [619].log_data[1].valid := 1, [619].log_data[2].valid := 1, [619].log_data[3].valid := 1, [619].log_data[4].valid := 1, [619].log_data[5].valid := 1, [619].log_data[6].valid := 1, [619].log_data[7].valid := 1, [619].log_data[8].valid := 1, [619].log_data[9].valid := 1, [619].log_data[10].valid := 1, [619].log_data[11].valid := 1, [619].log_data[12].valid := 1, [619].log_data[13].valid := 1, [619].log_data[14].valid := 1, [619].log_data[15].valid := 1, [619].log_data[16].valid := 1, [619].log_data[17].valid := 1, [619].log_data[18].valid := 1, [619].log_data[19].valid := 1, [619].time.Year := 2023, [619].time.Month := 1, [619].time.Day := 14, [619].time.Hour := 3, [619].time.Minute := 14, [619].time.Second := 59, [620].log_data[0].min := 1.0, [620].log_data[0].max := 1.0, [620].log_data[0].total := 900.0,
        [620].log_data[0].time := 900.0, [620].log_data[0].minminute := 15, [620].log_data[0].maxminute := 15, [620].log_data[0].valid := 1, [620].log_data[1].valid := 1, [620].log_data[2].valid := 1, [620].log_data[3].valid := 1, [620].log_data[4].valid := 1, [620].log_data[5].valid := 1, [620].log_data[6].valid := 1, [620].log_data[7].valid := 1, [620].log_data[8].valid := 1, [620].log_data[9].valid := 1, [620].log_data[10].valid := 1, [620].log_data[11].valid := 1, [620].log_data[12].valid := 1, [620].log_data[13].valid := 1, [620].log_data[14].valid := 1, [620].log_data[15].valid := 1, [620].log_data[16].valid := 1, [620].log_data[17].valid := 1, [620].log_data[18].valid := 1, [620].log_data[19].valid := 1, [620].time.Year := 2023, [620].time.Month := 1, [620].time.Day := 14, [620].time.Hour := 3, [620].time.Minute := 29, [620].time.Second := 59, [621].log_data[0].min := 1.0, [621].log_data[0].max := 1.0, [621].log_data[0].total := 900.0, [621].log_data[0].time := 900.0, [621].log_data[0].minminute := 30, [621].log_data[0].maxminute := 30, [621].log_data[0].valid := 1, [621].log_data[1].valid := 1, [621].log_data[2].valid := 1, [621].log_data[3].valid := 1, [621].log_data[4].valid := 1, [621].log_data[5].valid := 1, [621].log_data[6].valid := 1, [621].log_data[7].valid := 1, [621].log_data[8].valid := 1, [621].log_data[9].valid := 1, [621].log_data[10].valid := 1, [621].log_data[11].valid := 1, [621].log_data[12].valid := 1, [621].log_data[13].valid := 1, [621].log_data[14].valid := 1, [621].log_data[15].valid := 1, [621].log_data[16].valid := 1, [621].log_data[17].valid := 1, [621].log_data[18].valid := 1, [621].log_data[19].valid := 1, [621].time.Year := 2023, [621].time.Month := 1, [621].time.Day := 14, [621].time.Hour := 3, [621].time.Minute := 44,
        [621].time.Second := 59, [622].log_data[0].min := 1.0, [622].log_data[0].max := 1.0, [622].log_data[0].total := 900.0, [622].log_data[0].time := 900.0, [622].log_data[0].minminute := 45, [622].log_data[0].maxminute := 45, [622].log_data[0].valid := 1, [622].log_data[1].valid := 1, [622].log_data[2].valid := 1, [622].log_data[3].valid := 1, [622].log_data[4].valid := 1, [622].log_data[5].valid := 1, [622].log_data[6].valid := 1, [622].log_data[7].valid := 1, [622].log_data[8].valid := 1, [622].log_data[9].valid := 1, [622].log_data[10].valid := 1, [622].log_data[11].valid := 1, [622].log_data[12].valid := 1, [622].log_data[13].valid := 1, [622].log_data[14].valid := 1, [622].log_data[15].valid := 1, [622].log_data[16].valid := 1, [622].log_data[17].valid := 1, [622].log_data[18].valid := 1, [622].log_data[19].valid := 1, [622].time.Year := 2023, [622].time.Month := 1, [622].time.Day := 14, [622].time.Hour := 3, [622].time.Minute := 59, [622].time.Second := 59, [623].log_data[0].min := 1.0, [623].log_data[0].max := 1.0, [623].log_data[0].total := 900.0, [623].log_data[0].time := 900.0, [623].log_data[0].valid := 1, [623].log_data[1].valid := 1, [623].log_data[2].valid := 1, [623].log_data[3].valid := 1, [623].log_data[4].valid := 1, [623].log_data[5].valid := 1, [623].log_data[6].valid := 1, [623].log_data[7].valid := 1, [623].log_data[8].valid := 1, [623].log_data[9].valid := 1, [623].log_data[10].valid := 1, [623].log_data[11].valid := 1, [623].log_data[12].valid := 1, [623].log_data[13].valid := 1, [623].log_data[14].valid := 1, [623].log_data[15].valid := 1, [623].log_data[16].valid := 1, [623].log_data[17].valid := 1, [623].log_data[18].valid := 1, [623].log_data[19].valid := 1, [623].time.Year := 2023, [623].time.Month := 1, [623].time.Day := 14,
        [623].time.Hour := 4, [623].time.Minute := 14, [623].time.Second := 59, [624].log_data[0].min := 1.0, [624].log_data[0].max := 1.0, [624].log_data[0].total := 900.0, [624].log_data[0].time := 900.0, [624].log_data[0].minminute := 15, [624].log_data[0].maxminute := 15, [624].log_data[0].valid := 1, [624].log_data[1].valid := 1, [624].log_data[2].valid := 1, [624].log_data[3].valid := 1, [624].log_data[4].valid := 1, [624].log_data[5].valid := 1, [624].log_data[6].valid := 1, [624].log_data[7].valid := 1, [624].log_data[8].valid := 1, [624].log_data[9].valid := 1, [624].log_data[10].valid := 1, [624].log_data[11].valid := 1, [624].log_data[12].valid := 1, [624].log_data[13].valid := 1, [624].log_data[14].valid := 1, [624].log_data[15].valid := 1, [624].log_data[16].valid := 1, [624].log_data[17].valid := 1, [624].log_data[18].valid := 1, [624].log_data[19].valid := 1, [624].time.Year := 2023, [624].time.Month := 1, [624].time.Day := 14, [624].time.Hour := 4, [624].time.Minute := 29, [624].time.Second := 59, [625].log_data[0].min := 1.0, [625].log_data[0].max := 1.0, [625].log_data[0].total := 900.0, [625].log_data[0].time := 900.0, [625].log_data[0].minminute := 30, [625].log_data[0].maxminute := 30, [625].log_data[0].valid := 1, [625].log_data[1].valid := 1, [625].log_data[2].valid := 1, [625].log_data[3].valid := 1, [625].log_data[4].valid := 1, [625].log_data[5].valid := 1, [625].log_data[6].valid := 1, [625].log_data[7].valid := 1, [625].log_data[8].valid := 1, [625].log_data[9].valid := 1, [625].log_data[10].valid := 1, [625].log_data[11].valid := 1, [625].log_data[12].valid := 1, [625].log_data[13].valid := 1, [625].log_data[14].valid := 1, [625].log_data[15].valid := 1, [625].log_data[16].valid := 1, [625].log_data[17].valid := 1, [625].log_data[18].valid := 1,
        [625].log_data[19].valid := 1, [625].time.Year := 2023, [625].time.Month := 1, [625].time.Day := 14, [625].time.Hour := 4, [625].time.Minute := 44, [625].time.Second := 59, [626].log_data[0].min := 1.0, [626].log_data[0].max := 1.0, [626].log_data[0].total := 900.0, [626].log_data[0].time := 900.0, [626].log_data[0].minminute := 45, [626].log_data[0].maxminute := 45, [626].log_data[0].valid := 1, [626].log_data[1].valid := 1, [626].log_data[2].valid := 1, [626].log_data[3].valid := 1, [626].log_data[4].valid := 1, [626].log_data[5].valid := 1, [626].log_data[6].valid := 1, [626].log_data[7].valid := 1, [626].log_data[8].valid := 1, [626].log_data[9].valid := 1, [626].log_data[10].valid := 1, [626].log_data[11].valid := 1, [626].log_data[12].valid := 1, [626].log_data[13].valid := 1, [626].log_data[14].valid := 1, [626].log_data[15].valid := 1, [626].log_data[16].valid := 1, [626].log_data[17].valid := 1, [626].log_data[18].valid := 1, [626].log_data[19].valid := 1, [626].time.Year := 2023, [626].time.Month := 1, [626].time.Day := 14, [626].time.Hour := 4, [626].time.Minute := 59, [626].time.Second := 59, [627].log_data[0].min := 1.0, [627].log_data[0].max := 1.0, [627].log_data[0].total := 900.0, [627].log_data[0].time := 900.0, [627].log_data[0].valid := 1, [627].log_data[1].valid := 1, [627].log_data[2].valid := 1, [627].log_data[3].valid := 1, [627].log_data[4].valid := 1, [627].log_data[5].valid := 1, [627].log_data[6].valid := 1, [627].log_data[7].valid := 1, [627].log_data[8].valid := 1, [627].log_data[9].valid := 1, [627].log_data[10].valid := 1, [627].log_data[11].valid := 1, [627].log_data[12].valid := 1, [627].log_data[13].valid := 1, [627].log_data[14].valid := 1, [627].log_data[15].valid := 1, [627].log_data[16].valid := 1,
